LIN {X 0,Y 297.878,Z 251.743,A -85,B 0,C 180,E1 -16462.256,E2 -16462.256} C_VEL
LIN {X 0,Y 297.967,Z 251.372,A -85,B 0,C 180,E1 -16463.229,E2 -16463.229} C_VEL
LIN {X 0,Y 298.216,Z 251.337,A -85,B 0,C 180,E1 -16465.947,E2 -16465.947} C_VEL
LIN {X 0,Y 298.812,Z 251.261,A -85,B 0,C 180,E1 -16468.654,E2 -16468.654} C_VEL
LIN {X 0,Y 298.912,Z 251.253,A -85,B 0,C 180,E1 -16471.349,E2 -16471.349} C_VEL
LIN {X 0,Y 298.784,Z 251.266,A -85,B 0,C 180,E1 -16476.756,E2 -16476.756} C_VEL
LIN {X 0,Y 298.668,Z 251.281,A -85,B 0,C 180,E1 -16479.482,E2 -16479.482} C_VEL
LIN {X 0,Y 298.542,Z 251.295,A -85,B 0,C 180,E1 -16483.617,E2 -16483.617} C_VEL
LIN {X 0,Y 298.538,Z 251.296,A -85,B 0,C 180,E1 -16486.411,E2 -16486.411} C_VEL
LIN {X 0,Y 298.531,Z 251.297,A -85,B 0,C 180,E1 -16489.673,E2 -16489.673} C_VEL
LIN {X 0,Y 298.449,Z 251.307,A -85,B 0,C 180,E1 -16493.6,E2 -16493.6} C_VEL
LIN {X 0,Y 298.482,Z 251.306,A -85,B 0,C 180,E1 -16496.577,E2 -16496.577} C_VEL
LIN {X 0,Y 298.412,Z 251.312,A -85,B 0,C 180,E1 -16499.643,E2 -16499.643} C_VEL
LIN {X 0,Y 298.387,Z 251.319,A -85,B 0,C 180,E1 -16502.803,E2 -16502.803} C_VEL
LIN {X 0,Y 298.459,Z 251.309,A -85,B 0,C 180,E1 -16506.815,E2 -16506.815} C_VEL
LIN {X 0,Y 298.446,Z 251.307,A -85,B 0,C 180,E1 -16511.253,E2 -16511.253} C_VEL
LIN {X 0,Y 298.412,Z 251.311,A -85,B 0,C 180,E1 -16515.05,E2 -16515.05} C_VEL
LIN {X 0,Y 298.417,Z 251.313,A -85,B 0,C 180,E1 -16518.747,E2 -16518.747} C_VEL
LIN {X 0,Y 298.444,Z 251.309,A -85,B 0,C 180,E1 -16522.25,E2 -16522.25} C_VEL
LIN {X 0,Y 298.406,Z 251.307,A -85,B 0,C 180,E1 -16525.584,E2 -16525.584} C_VEL
LIN {X 0,Y 298.391,Z 251.314,A -85,B 0,C 180,E1 -16528.794,E2 -16528.794} C_VEL
LIN {X 0,Y 298.459,Z 251.307,A -85,B 0,C 180,E1 -16531.907,E2 -16531.907} C_VEL
LIN {X 0,Y 298.486,Z 251.301,A -85,B 0,C 180,E1 -16534.927,E2 -16534.927} C_VEL
LIN {X 0,Y 298.452,Z 251.301,A -85,B 0,C 180,E1 -16539.318,E2 -16539.318} C_VEL
LIN {X 0,Y 298.541,Z 251.297,A -85,B 0,C 180,E1 -16542.182,E2 -16542.182} C_VEL
LIN {X 0,Y 298.597,Z 251.287,A -85,B 0,C 180,E1 -16544.997,E2 -16544.997} C_VEL
LIN {X 0,Y 298.597,Z 251.287,A -85,B 0,C 180,E1 -16549.149,E2 -16549.149} C_VEL
LIN {X 0,Y 298.723,Z 251.274,A -85,B 0,C 180,E1 -16551.887,E2 -16551.887} C_VEL
LIN {X 0,Y 298.777,Z 251.262,A -85,B 0,C 180,E1 -16553.205,E2 -16553.205} C_VEL
LIN {X 0,Y 298.199,Z 251.337,A -85,B 0,C 180,E1 -16554.33,E2 -16554.33} C_VEL
LIN {X 0,Y 295.397,Z 251.687,A -85,B 0,C 180,E1 -16556.162,E2 -16556.162} C_VEL
LIN {X 0,Y 292.986,Z 251.988,A -85,B 0,C 180,E1 -16557.65,E2 -16557.65} C_VEL
LIN {X 0,Y 291.971,Z 252.112,A -85,B 0,C 180,E1 -16558.802,E2 -16558.802} C_VEL
LIN {X 0,Y 291.901,Z 252.12,A -85,B 0,C 180,E1 -16559.192,E2 -16559.192} C_VEL
LIN {X 0,Y 291.792,Z 252.135,A -85,B 0,C 180,E1 -16562.763,E2 -16562.763} C_VEL
LIN {X 0,Y 291.715,Z 252.142,A -85,B 0,C 180,E1 -16566.921,E2 -16566.921} C_VEL
LIN {X 0,Y 291.577,Z 252.165,A -85,B 0,C 180,E1 -16569.716,E2 -16569.716} C_VEL
LIN {X 0,Y 291.531,Z 252.17,A -85,B 0,C 180,E1 -16573.952,E2 -16573.952} C_VEL
LIN {X 0,Y 291.497,Z 252.172,A -85,B 0,C 180,E1 -16576.819,E2 -16576.819} C_VEL
LIN {X 0,Y 291.461,Z 252.177,A -85,B 0,C 180,E1 -16579.876,E2 -16579.876} C_VEL
LIN {X 0,Y 291.409,Z 252.183,A -85,B 0,C 180,E1 -16584.206,E2 -16584.206} C_VEL
LIN {X 0,Y 291.429,Z 252.183,A -85,B 0,C 180,E1 -16587.273,E2 -16587.273} C_VEL
LIN {X 0,Y 291.345,Z 252.191,A -85,B 0,C 180,E1 -16590.438,E2 -16590.438} C_VEL
LIN {X 0,Y 291.355,Z 252.191,A -85,B 0,C 180,E1 -16593.699,E2 -16593.699} C_VEL
LIN {X 0,Y 291.383,Z 252.19,A -85,B 0,C 180,E1 -16597.253,E2 -16597.253} C_VEL
LIN {X 0,Y 291.358,Z 252.193,A -85,B 0,C 180,E1 -16600.64,E2 -16600.64} C_VEL
LIN {X 0,Y 291.407,Z 252.343,A -85,B 0,C 180,E1 -16601.98,E2 -16601.98} C_VEL
LIN {X 0,Y 292.29,Z 257.456,A -85,B 0,C 180,E1 -16606.167,E2 -16606.167} C_VEL
LIN {X 0,Y 293.236,Z 262.543,A -85,B 0,C 180,E1 -16610.083,E2 -16610.083} C_VEL
LIN {X 0,Y 293.719,Z 266.92,A -85,B 0,C 180,E1 -16613.258,E2 -16613.258} C_VEL
LIN {X 0,Y 293.218,Z 270.535,A -85,B 0,C 180,E1 -16615.717,E2 -16615.717} C_VEL
LIN {X 0,Y 292.053,Z 277.114,A -85,B 0,C 180,E1 -16620.035,E2 -16620.035} C_VEL
LIN {X 0,Y 291.177,Z 283.685,A -85,B 0,C 180,E1 -16624.248,E2 -16624.248} C_VEL
LIN {X 0,Y 290.805,Z 286.658,A -85,B 0,C 180,E1 -16626.123,E2 -16626.123} C_VEL
LIN {X 0,Y 293.175,Z 300.593,A -85,B 0,C 180,E1 -16626.941,E2 -16626.941} C_VEL
LIN {X 0,Y 294.855,Z 313.515,A -85,B 0,C 180,E1 -16627.954,E2 -16627.954} C_VEL
LIN {X 0,Y 295.966,Z 325.481,A -85,B 0,C 180,E1 -16629.132,E2 -16629.132} C_VEL
LIN {X 0,Y 296.311,Z 334.899,A -85,B 0,C 180,E1 -16630.244,E2 -16630.244} C_VEL
LIN {X 0,Y 294.73,Z 346.056,A -85,B 0,C 180,E1 -16631.76,E2 -16631.76} C_VEL
LIN {X 0,Y 293.359,Z 355.626,A -85,B 0,C 180,E1 -16633.396,E2 -16633.396} C_VEL
LIN {X 0,Y 292.309,Z 363.424,A -85,B 0,C 180,E1 -16635.02,E2 -16635.02} C_VEL
LIN {X 0,Y 291.179,Z 371.571,A -85,B 0,C 180,E1 -16637.098,E2 -16637.098} C_VEL
LIN {X 0,Y 290.406,Z 377.096,A -85,B 0,C 180,E1 -16638.835,E2 -16638.835} C_VEL
LIN {X 0,Y 289.909,Z 382.504,A -85,B 0,C 180,E1 -16640.933,E2 -16640.933} C_VEL
LIN {X 0,Y 289.662,Z 386.705,A -85,B 0,C 180,E1 -16643.031,E2 -16643.031} C_VEL
LIN {X 0,Y 289.565,Z 388.913,A -85,B 0,C 180,E1 -16644.427,E2 -16644.427} C_VEL
LIN {X 0,Y 289.594,Z 390.629,A -85,B 0,C 180,E1 -16645.823,E2 -16645.823} C_VEL
LIN {X 0,Y 289.587,Z 391.918,A -85,B 0,C 180,E1 -16647.216,E2 -16647.216} C_VEL
LIN {X 0,Y 289.641,Z 392.803,A -85,B 0,C 180,E1 -16648.608,E2 -16648.608} C_VEL
LIN {X 0,Y 289.722,Z 393.271,A -85,B 0,C 180,E1 -16649.999,E2 -16649.999} C_VEL
LIN {X 0,Y 289.603,Z 393.288,A -85,B 0,C 180,E1 -16651.389,E2 -16651.389} C_VEL
LIN {X 0,Y 289.559,Z 392.914,A -85,B 0,C 180,E1 -16652.781,E2 -16652.781} C_VEL
LIN {X 0,Y 289.534,Z 392.146,A -85,B 0,C 180,E1 -16654.175,E2 -16654.175} C_VEL
LIN {X 0,Y 289.522,Z 390.972,A -85,B 0,C 180,E1 -16655.571,E2 -16655.571} C_VEL
LIN {X 0,Y 289.707,Z 388.403,A -85,B 0,C 180,E1 -16657.666,E2 -16657.666} C_VEL
LIN {X 0,Y 290.078,Z 384.831,A -85,B 0,C 180,E1 -16659.763,E2 -16659.763} C_VEL
LIN {X 0,Y 290.74,Z 380.19,A -85,B 0,C 180,E1 -16661.855,E2 -16661.855} C_VEL
LIN {X 0,Y 292.151,Z 373.245,A -85,B 0,C 180,E1 -16664.273,E2 -16664.273} C_VEL
LIN {X 0,Y 293.628,Z 365.768,A -85,B 0,C 180,E1 -16666.333,E2 -16666.333} C_VEL
LIN {X 0,Y 295.354,Z 356.558,A -85,B 0,C 180,E1 -16668.377,E2 -16668.377} C_VEL
LIN {X 0,Y 297.474,Z 346.002,A -85,B 0,C 180,E1 -16670.212,E2 -16670.212} C_VEL
LIN {X 0,Y 299.119,Z 336.644,A -85,B 0,C 180,E1 -16671.537,E2 -16671.537} C_VEL
LIN {X 0,Y 299.097,Z 325.654,A -85,B 0,C 180,E1 -16672.954,E2 -16672.954} C_VEL
LIN {X 0,Y 298.03,Z 313.134,A -85,B 0,C 180,E1 -16674.348,E2 -16674.348} C_VEL
LIN {X 0,Y 295.882,Z 300.736,A -85,B 0,C 180,E1 -16675.557,E2 -16675.557} C_VEL
LIN {X 0,Y 292.49,Z 287.558,A -85,B 0,C 180,E1 -16676.695,E2 -16676.695} C_VEL
LIN {X 0,Y 291.601,Z 284.162,A -85,B 0,C 180,E1 -16676.947,E2 -16676.947} C_VEL
LIN {X 0,Y 292.841,Z 276.861,A -85,B 0,C 180,E1 -16681.868,E2 -16681.868} C_VEL
LIN {X 0,Y 293.931,Z 271.595,A -85,B 0,C 180,E1 -16685.612,E2 -16685.612} C_VEL
LIN {X 0,Y 294.175,Z 270.188,A -85,B 0,C 180,E1 -16686.672,E2 -16686.672} C_VEL
LIN {X 0,Y 294.068,Z 267.992,A -85,B 0,C 180,E1 -16688.415,E2 -16688.415} C_VEL
LIN {X 0,Y 293.408,Z 263.727,A -85,B 0,C 180,E1 -16692.118,E2 -16692.118} C_VEL
LIN {X 0,Y 292.651,Z 259.608,A -85,B 0,C 180,E1 -16696.089,E2 -16696.089} C_VEL
LIN {X 0,Y 291.977,Z 255.678,A -85,B 0,C 180,E1 -16700.374,E2 -16700.374} C_VEL
LIN {X 0,Y 291.629,Z 253.619,A -85,B 0,C 180,E1 -16702.95,E2 -16702.95} C_VEL
LIN {X 0,Y 291.369,Z 252.194,A -85,B 0,C 180,E1 -16705.092,E2 -16705.092} C_VEL
LIN {X 0,Y 291.371,Z 252.194,A -85,B 0,C 180,E1 -16707.949,E2 -16707.949} C_VEL
LIN {X 0,Y 291.38,Z 252.191,A -85,B 0,C 180,E1 -16711.156,E2 -16711.156} C_VEL
LIN {X 0,Y 291.414,Z 252.187,A -85,B 0,C 180,E1 -16714.27,E2 -16714.27} C_VEL
LIN {X 0,Y 291.379,Z 252.19,A -85,B 0,C 180,E1 -16717.297,E2 -16717.297} C_VEL
LIN {X 0,Y 291.455,Z 252.18,A -85,B 0,C 180,E1 -16720.268,E2 -16720.268} C_VEL
LIN {X 0,Y 291.551,Z 252.168,A -85,B 0,C 180,E1 -16724.621,E2 -16724.621} C_VEL
LIN {X 0,Y 291.534,Z 252.171,A -85,B 0,C 180,E1 -16728.878,E2 -16728.878} C_VEL
LIN {X 0,Y 291.704,Z 252.15,A -85,B 0,C 180,E1 -16731.686,E2 -16731.686} C_VEL
LIN {X 0,Y 291.627,Z 252.159,A -85,B 0,C 180,E1 -16734.466,E2 -16734.466} C_VEL
LIN {X 0,Y 291.884,Z 252.128,A -85,B 0,C 180,E1 -16738.618,E2 -16738.618} C_VEL
LIN {X 0,Y 291.885,Z 252.128,A -85,B 0,C 180,E1 -16741.378,E2 -16741.378} C_VEL
LIN {X 0,Y 291.739,Z 252.143,A -85,B 0,C 180,E1 -16746.916,E2 -16746.916} C_VEL
LIN {X 0,Y 291.621,Z 252.162,A -85,B 0,C 180,E1 -16749.71,E2 -16749.71} C_VEL
LIN {X 0,Y 291.504,Z 252.179,A -85,B 0,C 180,E1 -16753.949,E2 -16753.949} C_VEL
LIN {X 0,Y 291.548,Z 253.73,A -85,B 0,C 180,E1 -16756.812,E2 -16756.812} C_VEL
LIN {X 0,Y 291.501,Z 255.573,A -85,B 0,C 180,E1 -16759.906,E2 -16759.906} C_VEL
LIN {X 0,Y 291.255,Z 257.883,A -85,B 0,C 180,E1 -16763.521,E2 -16763.521} C_VEL
LIN {X 0,Y 291.048,Z 259.624,A -85,B 0,C 180,E1 -16766.095,E2 -16766.095} C_VEL
LIN {X 0,Y 292.201,Z 262.851,A -85,B 0,C 180,E1 -16766.414,E2 -16766.414} C_VEL
LIN {X 0,Y 296.691,Z 274.182,A -85,B 0,C 180,E1 -16767.651,E2 -16767.651} C_VEL
LIN {X 0,Y 299.912,Z 284.645,A -85,B 0,C 180,E1 -16768.88,E2 -16768.88} C_VEL
LIN {X 0,Y 302.255,Z 295.27,A -85,B 0,C 180,E1 -16770.242,E2 -16770.242} C_VEL
LIN {X 0,Y 302.598,Z 297.676,A -85,B 0,C 180,E1 -16770.569,E2 -16770.569} C_VEL
LIN {X 0,Y 300.991,Z 308.423,A -85,B 0,C 180,E1 -16771.863,E2 -16771.863} C_VEL
LIN {X 0,Y 299.09,Z 319.099,A -85,B 0,C 180,E1 -16773.472,E2 -16773.472} C_VEL
LIN {X 0,Y 297.172,Z 328.8,A -85,B 0,C 180,E1 -16775.325,E2 -16775.325} C_VEL
LIN {X 0,Y 295.453,Z 336.613,A -85,B 0,C 180,E1 -16777.17,E2 -16777.17} C_VEL
LIN {X 0,Y 293.915,Z 343.386,A -85,B 0,C 180,E1 -16779.153,E2 -16779.153} C_VEL
LIN {X 0,Y 292.712,Z 348.623,A -85,B 0,C 180,E1 -16781.07,E2 -16781.07} C_VEL
LIN {X 0,Y 291.737,Z 352.849,A -85,B 0,C 180,E1 -16783.018,E2 -16783.018} C_VEL
LIN {X 0,Y 290.734,Z 356.874,A -85,B 0,C 180,E1 -16785.493,E2 -16785.493} C_VEL
LIN {X 0,Y 290.171,Z 358.907,A -85,B 0,C 180,E1 -16787.302,E2 -16787.302} C_VEL
LIN {X 0,Y 289.823,Z 360.236,A -85,B 0,C 180,E1 -16789.103,E2 -16789.103} C_VEL
LIN {X 0,Y 289.581,Z 360.934,A -85,B 0,C 180,E1 -16790.948,E2 -16790.948} C_VEL
LIN {X 0,Y 289.434,Z 360.798,A -85,B 0,C 180,E1 -16793.25,E2 -16793.25} C_VEL
LIN {X 0,Y 289.574,Z 359.526,A -85,B 0,C 180,E1 -16795.602,E2 -16795.602} C_VEL
LIN {X 0,Y 289.895,Z 356.973,A -85,B 0,C 180,E1 -16798.045,E2 -16798.045} C_VEL
LIN {X 0,Y 290.474,Z 352.938,A -85,B 0,C 180,E1 -16800.571,E2 -16800.571} C_VEL
LIN {X 0,Y 291.068,Z 348.315,A -85,B 0,C 180,E1 -16802.694,E2 -16802.694} C_VEL
LIN {X 0,Y 291.918,Z 342.744,A -85,B 0,C 180,E1 -16804.703,E2 -16804.703} C_VEL
LIN {X 0,Y 292.962,Z 335.902,A -85,B 0,C 180,E1 -16806.684,E2 -16806.684} C_VEL
LIN {X 0,Y 294.217,Z 327.347,A -85,B 0,C 180,E1 -16808.677,E2 -16808.677} C_VEL
LIN {X 0,Y 295.76,Z 317.21,A -85,B 0,C 180,E1 -16810.57,E2 -16810.57} C_VEL
LIN {X 0,Y 297.122,Z 306.976,A -85,B 0,C 180,E1 -16812.093,E2 -16812.093} C_VEL
LIN {X 0,Y 298.379,Z 295.987,A -85,B 0,C 180,E1 -16813.407,E2 -16813.407} C_VEL
LIN {X 0,Y 298.756,Z 292.354,A -85,B 0,C 180,E1 -16813.78,E2 -16813.78} C_VEL
LIN {X 0,Y 296.429,Z 280.089,A -85,B 0,C 180,E1 -16815.065,E2 -16815.065} C_VEL
LIN {X 0,Y 293.36,Z 267.572,A -85,B 0,C 180,E1 -16816.14,E2 -16816.14} C_VEL
LIN {X 0,Y 290.474,Z 257.017,A -85,B 0,C 180,E1 -16816.891,E2 -16816.891} C_VEL
LIN {X 0,Y 290.734,Z 253.095,A -85,B 0,C 180,E1 -16821.662,E2 -16821.662} C_VEL
LIN {X 0,Y 290.89,Z 252.254,A -85,B 0,C 180,E1 -16823.063,E2 -16823.063} C_VEL
LIN {X 0,Y 291.164,Z 252.216,A -85,B 0,C 180,E1 -16825.849,E2 -16825.849} C_VEL
LIN {X 0,Y 291.768,Z 252.139,A -85,B 0,C 180,E1 -16828.621,E2 -16828.621} C_VEL
LIN {X 0,Y 291.878,Z 252.129,A -85,B 0,C 180,E1 -16831.381,E2 -16831.381} C_VEL
LIN {X 0,Y 291.733,Z 252.145,A -85,B 0,C 180,E1 -16836.92,E2 -16836.92} C_VEL
LIN {X 0,Y 291.617,Z 252.158,A -85,B 0,C 180,E1 -16839.714,E2 -16839.714} C_VEL
LIN {X 0,Y 291.511,Z 252.169,A -85,B 0,C 180,E1 -16843.952,E2 -16843.952} C_VEL
LIN {X 0,Y 291.477,Z 252.178,A -85,B 0,C 180,E1 -16846.82,E2 -16846.82} C_VEL
LIN {X 0,Y 291.473,Z 252.176,A -85,B 0,C 180,E1 -16849.895,E2 -16849.895} C_VEL
LIN {X 0,Y 291.392,Z 252.186,A -85,B 0,C 180,E1 -16854.207,E2 -16854.207} C_VEL
LIN {X 0,Y 291.416,Z 252.185,A -85,B 0,C 180,E1 -16857.274,E2 -16857.274} C_VEL
LIN {X 0,Y 291.329,Z 252.196,A -85,B 0,C 180,E1 -16860.439,E2 -16860.439} C_VEL
LIN {X 0,Y 291.337,Z 252.192,A -85,B 0,C 180,E1 -16863.701,E2 -16863.701} C_VEL
LIN {X 0,Y 291.392,Z 252.187,A -85,B 0,C 180,E1 -16867.263,E2 -16867.263} C_VEL
LIN {X 0,Y 291.395,Z 252.189,A -85,B 0,C 180,E1 -16870.634,E2 -16870.634} C_VEL
LIN {X 0,Y 291.348,Z 252.194,A -85,B 0,C 180,E1 -16874.393,E2 -16874.393} C_VEL
LIN {X 0,Y 291.354,Z 252.194,A -85,B 0,C 180,E1 -16878.4,E2 -16878.4} C_VEL
LIN {X 0,Y 291.378,Z 252.186,A -85,B 0,C 180,E1 -16881.166,E2 -16881.166} C_VEL
LIN {X 0,Y 291.384,Z 252.183,A -85,B 0,C 180,E1 -16884.633,E2 -16884.633} C_VEL
LIN {X 0,Y 291.369,Z 252.187,A -85,B 0,C 180,E1 -16887.953,E2 -16887.953} C_VEL
LIN {X 0,Y 291.377,Z 252.187,A -85,B 0,C 180,E1 -16891.161,E2 -16891.161} C_VEL
LIN {X 0,Y 291.416,Z 252.186,A -85,B 0,C 180,E1 -16894.275,E2 -16894.275} C_VEL
LIN {X 0,Y 291.383,Z 252.184,A -85,B 0,C 180,E1 -16897.302,E2 -16897.302} C_VEL
LIN {X 0,Y 291.461,Z 252.176,A -85,B 0,C 180,E1 -16900.273,E2 -16900.273} C_VEL
LIN {X 0,Y 291.559,Z 252.165,A -85,B 0,C 180,E1 -16904.626,E2 -16904.626} C_VEL
LIN {X 0,Y 291.541,Z 252.166,A -85,B 0,C 180,E1 -16908.883,E2 -16908.883} C_VEL
LIN {X 0,Y 291.673,Z 252.152,A -85,B 0,C 180,E1 -16911.69,E2 -16911.69} C_VEL
LIN {X 0,Y 291.629,Z 252.151,A -85,B 0,C 180,E1 -16914.471,E2 -16914.471} C_VEL
LIN {X 0,Y 291.895,Z 252.122,A -85,B 0,C 180,E1 -16918.623,E2 -16918.623} C_VEL
LIN {X 0,Y 291.901,Z 252.12,A -85,B 0,C 180,E1 -16919.192,E2 -16919.192} C_VEL
LIN {X 0,Y 291.59,Z 252.164,A -85,B 0,C 180,E1 -16919.962,E2 -16919.962} C_VEL
LIN {X 0,Y 290.177,Z 252.339,A -85,B 0,C 180,E1 -16921.096,E2 -16921.096} C_VEL
LIN {X 0,Y 285.646,Z 252.904,A -85,B 0,C 180,E1 -16923.731,E2 -16923.731} C_VEL
LIN {X 0,Y 284.607,Z 253.029,A -85,B 0,C 180,E1 -16924.912,E2 -16924.912} C_VEL
LIN {X 0,Y 284.553,Z 253.035,A -85,B 0,C 180,E1 -16925.312,E2 -16925.312} C_VEL
LIN {X 0,Y 284.63,Z 253.024,A -85,B 0,C 180,E1 -16928.522,E2 -16928.522} C_VEL
LIN {X 0,Y 284.484,Z 253.046,A -85,B 0,C 180,E1 -16932.849,E2 -16932.849} C_VEL
LIN {X 0,Y 284.497,Z 253.046,A -85,B 0,C 180,E1 -16935.77,E2 -16935.77} C_VEL
LIN {X 0,Y 284.389,Z 253.056,A -85,B 0,C 180,E1 -16940.244,E2 -16940.244} C_VEL
LIN {X 0,Y 284.379,Z 253.06,A -85,B 0,C 180,E1 -16943.876,E2 -16943.876} C_VEL
LIN {X 0,Y 284.405,Z 253.058,A -85,B 0,C 180,E1 -16947.173,E2 -16947.173} C_VEL
LIN {X 0,Y 284.304,Z 253.073,A -85,B 0,C 180,E1 -16951.275,E2 -16951.275} C_VEL
LIN {X 0,Y 284.351,Z 253.065,A -85,B 0,C 180,E1 -16955.349,E2 -16955.349} C_VEL
LIN {X 0,Y 284.319,Z 253.066,A -85,B 0,C 180,E1 -16958.17,E2 -16958.17} C_VEL
LIN {X 0,Y 284.37,Z 253.201,A -85,B 0,C 180,E1 -16961.623,E2 -16961.623} C_VEL
LIN {X 0,Y 285.156,Z 257.944,A -85,B 0,C 180,E1 -16965.624,E2 -16965.624} C_VEL
LIN {X 0,Y 286.115,Z 262.952,A -85,B 0,C 180,E1 -16969.596,E2 -16969.596} C_VEL
LIN {X 0,Y 286.675,Z 267.618,A -85,B 0,C 180,E1 -16973.083,E2 -16973.083} C_VEL
LIN {X 0,Y 286.2,Z 271.238,A -85,B 0,C 180,E1 -16975.61,E2 -16975.61} C_VEL
LIN {X 0,Y 284.88,Z 278.396,A -85,B 0,C 180,E1 -16980.434,E2 -16980.434} C_VEL
LIN {X 0,Y 284.065,Z 284.332,A -85,B 0,C 180,E1 -16984.343,E2 -16984.343} C_VEL
LIN {X 0,Y 283.82,Z 286.254,A -85,B 0,C 180,E1 -16985.591,E2 -16985.591} C_VEL
LIN {X 0,Y 286.285,Z 300.737,A -85,B 0,C 180,E1 -16986.494,E2 -16986.494} C_VEL
LIN {X 0,Y 288.003,Z 314.305,A -85,B 0,C 180,E1 -16987.606,E2 -16987.606} C_VEL
LIN {X 0,Y 289.03,Z 325.864,A -85,B 0,C 180,E1 -16988.794,E2 -16988.794} C_VEL
LIN {X 0,Y 289.403,Z 335.147,A -85,B 0,C 180,E1 -16989.938,E2 -16989.938} C_VEL
LIN {X 0,Y 287.773,Z 346.146,A -85,B 0,C 180,E1 -16991.488,E2 -16991.488} C_VEL
LIN {X 0,Y 286.353,Z 355.715,A -85,B 0,C 180,E1 -16993.178,E2 -16993.178} C_VEL
LIN {X 0,Y 285.156,Z 364.113,A -85,B 0,C 180,E1 -16995.001,E2 -16995.001} C_VEL
LIN {X 0,Y 284.036,Z 372.066,A -85,B 0,C 180,E1 -16997.131,E2 -16997.131} C_VEL
LIN {X 0,Y 283.186,Z 378.4,A -85,B 0,C 180,E1 -16999.271,E2 -16999.271} C_VEL
LIN {X 0,Y 282.756,Z 383.437,A -85,B 0,C 180,E1 -17001.422,E2 -17001.422} C_VEL
LIN {X 0,Y 282.538,Z 387.312,A -85,B 0,C 180,E1 -17003.572,E2 -17003.572} C_VEL
LIN {X 0,Y 282.508,Z 390.131,A -85,B 0,C 180,E1 -17005.719,E2 -17005.719} C_VEL
LIN {X 0,Y 282.512,Z 391.443,A -85,B 0,C 180,E1 -17007.147,E2 -17007.147} C_VEL
LIN {X 0,Y 282.552,Z 392.348,A -85,B 0,C 180,E1 -17008.573,E2 -17008.573} C_VEL
LIN {X 0,Y 282.632,Z 392.851,A -85,B 0,C 180,E1 -17009.999,E2 -17009.999} C_VEL
LIN {X 0,Y 282.516,Z 392.895,A -85,B 0,C 180,E1 -17011.424,E2 -17011.424} C_VEL
LIN {X 0,Y 282.483,Z 392.541,A -85,B 0,C 180,E1 -17012.851,E2 -17012.851} C_VEL
LIN {X 0,Y 282.428,Z 390.827,A -85,B 0,C 180,E1 -17015.502,E2 -17015.502} C_VEL
LIN {X 0,Y 282.638,Z 388.111,A -85,B 0,C 180,E1 -17017.859,E2 -17017.859} C_VEL
LIN {X 0,Y 283.061,Z 384.593,A -85,B 0,C 180,E1 -17020.007,E2 -17020.007} C_VEL
LIN {X 0,Y 283.762,Z 380.014,A -85,B 0,C 180,E1 -17022.151,E2 -17022.151} C_VEL
LIN {X 0,Y 285.265,Z 373.162,A -85,B 0,C 180,E1 -17024.626,E2 -17024.626} C_VEL
LIN {X 0,Y 286.813,Z 365.752,A -85,B 0,C 180,E1 -17026.732,E2 -17026.732} C_VEL
LIN {X 0,Y 288.603,Z 356.636,A -85,B 0,C 180,E1 -17028.822,E2 -17028.822} C_VEL
LIN {X 0,Y 290.821,Z 346.209,A -85,B 0,C 180,E1 -17030.696,E2 -17030.696} C_VEL
LIN {X 0,Y 292.377,Z 338.261,A -85,B 0,C 180,E1 -17031.873,E2 -17031.873} C_VEL
LIN {X 0,Y 292.578,Z 328.257,A -85,B 0,C 180,E1 -17033.249,E2 -17033.249} C_VEL
LIN {X 0,Y 291.762,Z 315.977,A -85,B 0,C 180,E1 -17034.721,E2 -17034.721} C_VEL
LIN {X 0,Y 289.917,Z 304.046,A -85,B 0,C 180,E1 -17035.982,E2 -17035.982} C_VEL
LIN {X 0,Y 286.778,Z 290.743,A -85,B 0,C 180,E1 -17037.233,E2 -17037.233} C_VEL
LIN {X 0,Y 284.767,Z 284.329,A -85,B 0,C 180,E1 -17037.8,E2 -17037.8} C_VEL
LIN {X 0,Y 284.701,Z 283.664,A -85,B 0,C 180,E1 -17037.859,E2 -17037.859} C_VEL
LIN {X 0,Y 286.016,Z 276.704,A -85,B 0,C 180,E1 -17042.722,E2 -17042.722} C_VEL
LIN {X 0,Y 287.007,Z 272.147,A -85,B 0,C 180,E1 -17046.089,E2 -17046.089} C_VEL
LIN {X 0,Y 287.143,Z 270.064,A -85,B 0,C 180,E1 -17047.724,E2 -17047.724} C_VEL
LIN {X 0,Y 286.555,Z 265.789,A -85,B 0,C 180,E1 -17051.466,E2 -17051.466} C_VEL
LIN {X 0,Y 285.782,Z 261.651,A -85,B 0,C 180,E1 -17055.491,E2 -17055.491} C_VEL
LIN {X 0,Y 285.334,Z 259.033,A -85,B 0,C 180,E1 -17058.313,E2 -17058.313} C_VEL
LIN {X 0,Y 284.836,Z 255.837,A -85,B 0,C 180,E1 -17062.142,E2 -17062.142} C_VEL
LIN {X 0,Y 284.39,Z 253.529,A -85,B 0,C 180,E1 -17065.36,E2 -17065.36} C_VEL
LIN {X 0,Y 284.307,Z 253.073,A -85,B 0,C 180,E1 -17067.187,E2 -17067.187} C_VEL
LIN {X 0,Y 284.357,Z 253.067,A -85,B 0,C 180,E1 -17070.374,E2 -17070.374} C_VEL
LIN {X 0,Y 284.376,Z 253.063,A -85,B 0,C 180,E1 -17073.584,E2 -17073.584} C_VEL
LIN {X 0,Y 284.364,Z 253.066,A -85,B 0,C 180,E1 -17076.705,E2 -17076.705} C_VEL
LIN {X 0,Y 284.4,Z 253.059,A -85,B 0,C 180,E1 -17081.259,E2 -17081.259} C_VEL
LIN {X 0,Y 284.488,Z 253.047,A -85,B 0,C 180,E1 -17084.457,E2 -17084.457} C_VEL
LIN {X 0,Y 284.486,Z 253.048,A -85,B 0,C 180,E1 -17088.599,E2 -17088.599} C_VEL
LIN {X 0,Y 284.654,Z 253.028,A -85,B 0,C 180,E1 -17091.479,E2 -17091.479} C_VEL
LIN {X 0,Y 284.597,Z 253.035,A -85,B 0,C 180,E1 -17094.329,E2 -17094.329} C_VEL
LIN {X 0,Y 284.85,Z 253.004,A -85,B 0,C 180,E1 -17098.584,E2 -17098.584} C_VEL
LIN {X 0,Y 284.851,Z 253.004,A -85,B 0,C 180,E1 -17101.412,E2 -17101.412} C_VEL
LIN {X 0,Y 284.691,Z 253.021,A -85,B 0,C 180,E1 -17107.088,E2 -17107.088} C_VEL
LIN {X 0,Y 284.559,Z 253.04,A -85,B 0,C 180,E1 -17109.953,E2 -17109.953} C_VEL
LIN {X 0,Y 284.465,Z 253.053,A -85,B 0,C 180,E1 -17112.845,E2 -17112.845} C_VEL
LIN {X 0,Y 284.56,Z 254.408,A -85,B 0,C 180,E1 -17115.761,E2 -17115.761} C_VEL
LIN {X 0,Y 284.554,Z 256.055,A -85,B 0,C 180,E1 -17118.726,E2 -17118.726} C_VEL
LIN {X 0,Y 284.335,Z 257.92,A -85,B 0,C 180,E1 -17121.76,E2 -17121.76} C_VEL
LIN {X 0,Y 284.082,Z 260.226,A -85,B 0,C 180,E1 -17125.21,E2 -17125.21} C_VEL
LIN {X 0,Y 285.279,Z 263.405,A -85,B 0,C 180,E1 -17125.536,E2 -17125.536} C_VEL
LIN {X 0,Y 289.603,Z 273.829,A -85,B 0,C 180,E1 -17126.761,E2 -17126.761} C_VEL
LIN {X 0,Y 293.122,Z 284.677,A -85,B 0,C 180,E1 -17128.103,E2 -17128.103} C_VEL
LIN {X 0,Y 295.569,Z 295.709,A -85,B 0,C 180,E1 -17129.561,E2 -17129.561} C_VEL
LIN {X 0,Y 296.129,Z 299.137,A -85,B 0,C 180,E1 -17130.053,E2 -17130.053} C_VEL
LIN {X 0,Y 294.431,Z 309.949,A -85,B 0,C 180,E1 -17131.414,E2 -17131.414} C_VEL
LIN {X 0,Y 292.43,Z 320.362,A -85,B 0,C 180,E1 -17133.06,E2 -17133.06} C_VEL
LIN {X 0,Y 290.435,Z 329.954,A -85,B 0,C 180,E1 -17134.964,E2 -17134.964} C_VEL
LIN {X 0,Y 288.613,Z 337.763,A -85,B 0,C 180,E1 -17136.88,E2 -17136.88} C_VEL
LIN {X 0,Y 286.847,Z 344.951,A -85,B 0,C 180,E1 -17139.111,E2 -17139.111} C_VEL
LIN {X 0,Y 285.284,Z 351.331,A -85,B 0,C 180,E1 -17141.69,E2 -17141.69} C_VEL
LIN {X 0,Y 284.116,Z 355.828,A -85,B 0,C 180,E1 -17144.166,E2 -17144.166} C_VEL
LIN {X 0,Y 283.477,Z 358.296,A -85,B 0,C 180,E1 -17146.04,E2 -17146.04} C_VEL
LIN {X 0,Y 282.904,Z 360.21,A -85,B 0,C 180,E1 -17148.178,E2 -17148.178} C_VEL
LIN {X 0,Y 282.535,Z 361.253,A -85,B 0,C 180,E1 -17150.45,E2 -17150.45} C_VEL
LIN {X 0,Y 282.368,Z 361.142,A -85,B 0,C 180,E1 -17153.322,E2 -17153.322} C_VEL
LIN {X 0,Y 282.442,Z 360.211,A -85,B 0,C 180,E1 -17155.194,E2 -17155.194} C_VEL
LIN {X 0,Y 282.74,Z 357.885,A -85,B 0,C 180,E1 -17157.68,E2 -17157.68} C_VEL
LIN {X 0,Y 283.309,Z 354.064,A -85,B 0,C 180,E1 -17160.257,E2 -17160.257} C_VEL
LIN {X 0,Y 283.908,Z 349.509,A -85,B 0,C 180,E1 -17162.495,E2 -17162.495} C_VEL
LIN {X 0,Y 284.867,Z 343.382,A -85,B 0,C 180,E1 -17164.814,E2 -17164.814} C_VEL
LIN {X 0,Y 285.933,Z 336.614,A -85,B 0,C 180,E1 -17166.844,E2 -17166.844} C_VEL
LIN {X 0,Y 287.24,Z 328.14,A -85,B 0,C 180,E1 -17168.88,E2 -17168.88} C_VEL
LIN {X 0,Y 288.792,Z 318.404,A -85,B 0,C 180,E1 -17170.76,E2 -17170.76} C_VEL
LIN {X 0,Y 290.241,Z 307.938,A -85,B 0,C 180,E1 -17172.383,E2 -17172.383} C_VEL
LIN {X 0,Y 291.546,Z 297.063,A -85,B 0,C 180,E1 -17173.727,E2 -17173.727} C_VEL
LIN {X 0,Y 291.925,Z 293.518,A -85,B 0,C 180,E1 -17174.108,E2 -17174.108} C_VEL
LIN {X 0,Y 289.666,Z 281.484,A -85,B 0,C 180,E1 -17175.422,E2 -17175.422} C_VEL
LIN {X 0,Y 286.527,Z 268.683,A -85,B 0,C 180,E1 -17176.572,E2 -17176.572} C_VEL
LIN {X 0,Y 283.415,Z 257.418,A -85,B 0,C 180,E1 -17177.379,E2 -17177.379} C_VEL
LIN {X 0,Y 283.751,Z 253.539,A -85,B 0,C 180,E1 -17182.17,E2 -17182.17} C_VEL
LIN {X 0,Y 283.815,Z 253.136,A -85,B 0,C 180,E1 -17182.889,E2 -17182.889} C_VEL
LIN {X 0,Y 284.112,Z 253.095,A -85,B 0,C 180,E1 -17185.746,E2 -17185.746} C_VEL
LIN {X 0,Y 284.723,Z 253.016,A -85,B 0,C 180,E1 -17188.587,E2 -17188.587} C_VEL
LIN {X 0,Y 284.844,Z 253.005,A -85,B 0,C 180,E1 -17191.415,E2 -17191.415} C_VEL
LIN {X 0,Y 284.685,Z 253.025,A -85,B 0,C 180,E1 -17197.092,E2 -17197.092} C_VEL
LIN {X 0,Y 284.555,Z 253.037,A -85,B 0,C 180,E1 -17199.957,E2 -17199.957} C_VEL
LIN {X 0,Y 284.471,Z 253.046,A -85,B 0,C 180,E1 -17204.305,E2 -17204.305} C_VEL
LIN {X 0,Y 284.418,Z 253.059,A -85,B 0,C 180,E1 -17207.25,E2 -17207.25} C_VEL
LIN {X 0,Y 284.409,Z 253.056,A -85,B 0,C 180,E1 -17210.241,E2 -17210.241} C_VEL
LIN {X 0,Y 284.361,Z 253.062,A -85,B 0,C 180,E1 -17213.878,E2 -17213.878} C_VEL
LIN {X 0,Y 284.39,Z 253.061,A -85,B 0,C 180,E1 -17217.177,E2 -17217.177} C_VEL
LIN {X 0,Y 284.287,Z 253.073,A -85,B 0,C 180,E1 -17221.277,E2 -17221.277} C_VEL
LIN {X 0,Y 284.354,Z 253.063,A -85,B 0,C 180,E1 -17225.357,E2 -17225.357} C_VEL
LIN {X 0,Y 284.325,Z 253.067,A -85,B 0,C 180,E1 -17228.169,E2 -17228.169} C_VEL
LIN {X 0,Y 284.335,Z 253.066,A -85,B 0,C 180,E1 -17232.143,E2 -17232.143} C_VEL
LIN {X 0,Y 284.314,Z 253.068,A -85,B 0,C 180,E1 -17236.204,E2 -17236.204} C_VEL
LIN {X 0,Y 284.348,Z 253.064,A -85,B 0,C 180,E1 -17240.016,E2 -17240.016} C_VEL
LIN {X 0,Y 284.353,Z 253.059,A -85,B 0,C 180,E1 -17243.62,E2 -17243.62} C_VEL
LIN {X 0,Y 284.306,Z 253.064,A -85,B 0,C 180,E1 -17247.193,E2 -17247.193} C_VEL
LIN {X 0,Y 284.355,Z 253.066,A -85,B 0,C 180,E1 -17250.379,E2 -17250.379} C_VEL
LIN {X 0,Y 284.377,Z 253.06,A -85,B 0,C 180,E1 -17253.589,E2 -17253.589} C_VEL
LIN {X 0,Y 284.368,Z 253.058,A -85,B 0,C 180,E1 -17256.71,E2 -17256.71} C_VEL
LIN {X 0,Y 284.406,Z 253.05,A -85,B 0,C 180,E1 -17261.264,E2 -17261.264} C_VEL
LIN {X 0,Y 284.496,Z 253.045,A -85,B 0,C 180,E1 -17264.462,E2 -17264.462} C_VEL
LIN {X 0,Y 284.493,Z 253.045,A -85,B 0,C 180,E1 -17268.604,E2 -17268.604} C_VEL
LIN {X 0,Y 284.627,Z 253.027,A -85,B 0,C 180,E1 -17271.483,E2 -17271.483} C_VEL
LIN {X 0,Y 284.598,Z 253.027,A -85,B 0,C 180,E1 -17274.333,E2 -17274.333} C_VEL
LIN {X 0,Y 284.861,Z 252.998,A -85,B 0,C 180,E1 -17278.588,E2 -17278.588} C_VEL
LIN {X 0,Y 284.861,Z 253.001,A -85,B 0,C 180,E1 -17281.416,E2 -17281.416} C_VEL
LIN {X 0,Y 284.553,Z 253.035,A -85,B 0,C 180,E1 -17285.312,E2 -17285.312} C_VEL
LIN {X 0,Y 284.29,Z 253.071,A -85,B 0,C 180,E1 -17286.103,E2 -17286.103} C_VEL
LIN {X 0,Y 282.958,Z 253.236,A -85,B 0,C 180,E1 -17287.269,E2 -17287.269} C_VEL
LIN {X 0,Y 278.556,Z 253.785,A -85,B 0,C 180,E1 -17289.981,E2 -17289.981} C_VEL
LIN {X 0,Y 277.507,Z 253.915,A -85,B 0,C 180,E1 -17291.194,E2 -17291.194} C_VEL
LIN {X 0,Y 277.436,Z 253.927,A -85,B 0,C 180,E1 -17291.606,E2 -17291.606} C_VEL
LIN {X 0,Y 277.453,Z 253.923,A -85,B 0,C 180,E1 -17295.724,E2 -17295.724} C_VEL
LIN {X 0,Y 277.355,Z 253.932,A -85,B 0,C 180,E1 -17300.351,E2 -17300.351} C_VEL
LIN {X 0,Y 277.329,Z 253.938,A -85,B 0,C 180,E1 -17304.171,E2 -17304.171} C_VEL
LIN {X 0,Y 277.333,Z 253.937,A -85,B 0,C 180,E1 -17307.505,E2 -17307.505} C_VEL
LIN {X 0,Y 277.283,Z 253.943,A -85,B 0,C 180,E1 -17310.482,E2 -17310.482} C_VEL
LIN {X 0,Y 277.257,Z 253.946,A -85,B 0,C 180,E1 -17313.896,E2 -17313.896} C_VEL
LIN {X 0,Y 277.275,Z 253.946,A -85,B 0,C 180,E1 -17317.47,E2 -17317.47} C_VEL
LIN {X 0,Y 277.301,Z 254.025,A -85,B 0,C 180,E1 -17321.222,E2 -17321.222} C_VEL
LIN {X 0,Y 278.038,Z 258.43,A -85,B 0,C 180,E1 -17325.055,E2 -17325.055} C_VEL
LIN {X 0,Y 278.965,Z 263.364,A -85,B 0,C 180,E1 -17329.097,E2 -17329.097} C_VEL
LIN {X 0,Y 279.549,Z 267.195,A -85,B 0,C 180,E1 -17332.084,E2 -17332.084} C_VEL
LIN {X 0,Y 279.366,Z 270.698,A -85,B 0,C 180,E1 -17334.646,E2 -17334.646} C_VEL
LIN {X 0,Y 278.424,Z 275.472,A -85,B 0,C 180,E1 -17337.987,E2 -17337.987} C_VEL
LIN {X 0,Y 277.343,Z 282.061,A -85,B 0,C 180,E1 -17342.491,E2 -17342.491} C_VEL
LIN {X 0,Y 276.842,Z 285.927,A -85,B 0,C 180,E1 -17345.086,E2 -17345.086} C_VEL
LIN {X 0,Y 279.238,Z 299.838,A -85,B 0,C 180,E1 -17345.958,E2 -17345.958} C_VEL
LIN {X 0,Y 280.974,Z 312.957,A -85,B 0,C 180,E1 -17347.05,E2 -17347.05} C_VEL
LIN {X 0,Y 281.971,Z 324.437,A -85,B 0,C 180,E1 -17348.237,E2 -17348.237} C_VEL
LIN {X 0,Y 282.474,Z 335.386,A -85,B 0,C 180,E1 -17349.614,E2 -17349.614} C_VEL
LIN {X 0,Y 280.817,Z 346.234,A -85,B 0,C 180,E1 -17351.201,E2 -17351.201} C_VEL
LIN {X 0,Y 279.374,Z 355.725,A -85,B 0,C 180,E1 -17352.933,E2 -17352.933} C_VEL
LIN {X 0,Y 278.005,Z 364.797,A -85,B 0,C 180,E1 -17354.981,E2 -17354.981} C_VEL
LIN {X 0,Y 276.871,Z 372.491,A -85,B 0,C 180,E1 -17357.166,E2 -17357.166} C_VEL
LIN {X 0,Y 275.98,Z 379.582,A -85,B 0,C 180,E1 -17359.73,E2 -17359.73} C_VEL
LIN {X 0,Y 275.59,Z 384.28,A -85,B 0,C 180,E1 -17361.936,E2 -17361.936} C_VEL
LIN {X 0,Y 275.451,Z 388.095,A -85,B 0,C 180,E1 -17364.321,E2 -17364.321} C_VEL
LIN {X 0,Y 275.429,Z 389.635,A -85,B 0,C 180,E1 -17365.608,E2 -17365.608} C_VEL
LIN {X 0,Y 275.438,Z 390.968,A -85,B 0,C 180,E1 -17367.073,E2 -17367.073} C_VEL
LIN {X 0,Y 275.466,Z 391.894,A -85,B 0,C 180,E1 -17368.537,E2 -17368.537} C_VEL
LIN {X 0,Y 275.543,Z 392.421,A -85,B 0,C 180,E1 -17369.999,E2 -17369.999} C_VEL
LIN {X 0,Y 275.432,Z 392.503,A -85,B 0,C 180,E1 -17371.461,E2 -17371.461} C_VEL
LIN {X 0,Y 275.407,Z 392.169,A -85,B 0,C 180,E1 -17372.924,E2 -17372.924} C_VEL
LIN {X 0,Y 275.353,Z 390.323,A -85,B 0,C 180,E1 -17375.858,E2 -17375.858} C_VEL
LIN {X 0,Y 275.489,Z 388.779,A -85,B 0,C 180,E1 -17377.327,E2 -17377.327} C_VEL
LIN {X 0,Y 275.851,Z 385.657,A -85,B 0,C 180,E1 -17379.531,E2 -17379.531} C_VEL
LIN {X 0,Y 276.468,Z 381.496,A -85,B 0,C 180,E1 -17381.732,E2 -17381.732} C_VEL
LIN {X 0,Y 277.85,Z 375.176,A -85,B 0,C 180,E1 -17384.276,E2 -17384.276} C_VEL
LIN {X 0,Y 279.371,Z 368.35,A -85,B 0,C 180,E1 -17386.438,E2 -17386.438} C_VEL
LIN {X 0,Y 281.186,Z 359.976,A -85,B 0,C 180,E1 -17388.581,E2 -17388.581} C_VEL
LIN {X 0,Y 283.128,Z 351.445,A -85,B 0,C 180,E1 -17390.334,E2 -17390.334} C_VEL
LIN {X 0,Y 285.452,Z 341.014,A -85,B 0,C 180,E1 -17392.051,E2 -17392.051} C_VEL
LIN {X 0,Y 286.037,Z 333.671,A -85,B 0,C 180,E1 -17393.147,E2 -17393.147} C_VEL
LIN {X 0,Y 285.676,Z 321.895,A -85,B 0,C 180,E1 -17394.721,E2 -17394.721} C_VEL
LIN {X 0,Y 284.422,Z 310.182,A -85,B 0,C 180,E1 -17396.089,E2 -17396.089} C_VEL
LIN {X 0,Y 281.878,Z 297.338,A -85,B 0,C 180,E1 -17397.45,E2 -17397.45} C_VEL
LIN {X 0,Y 278.648,Z 286.404,A -85,B 0,C 180,E1 -17398.524,E2 -17398.524} C_VEL
LIN {X 0,Y 277.862,Z 283.15,A -85,B 0,C 180,E1 -17398.824,E2 -17398.824} C_VEL
LIN {X 0,Y 278.983,Z 277.664,A -85,B 0,C 180,E1 -17402.792,E2 -17402.792} C_VEL
LIN {X 0,Y 279.79,Z 274.342,A -85,B 0,C 180,E1 -17405.289,E2 -17405.289} C_VEL
LIN {X 0,Y 280.192,Z 272.142,A -85,B 0,C 180,E1 -17407.01,E2 -17407.01} C_VEL
LIN {X 0,Y 279.859,Z 268.908,A -85,B 0,C 180,E1 -17409.817,E2 -17409.817} C_VEL
LIN {X 0,Y 279.279,Z 265.397,A -85,B 0,C 180,E1 -17413.13,E2 -17413.13} C_VEL
LIN {X 0,Y 278.602,Z 261.634,A -85,B 0,C 180,E1 -17417.068,E2 -17417.068} C_VEL
LIN {X 0,Y 278.057,Z 258.467,A -85,B 0,C 180,E1 -17420.808,E2 -17420.808} C_VEL
LIN {X 0,Y 277.6,Z 255.818,A -85,B 0,C 180,E1 -17424.386,E2 -17424.386} C_VEL
LIN {X 0,Y 277.315,Z 254.287,A -85,B 0,C 180,E1 -17426.751,E2 -17426.751} C_VEL
LIN {X 0,Y 277.243,Z 253.954,A -85,B 0,C 180,E1 -17427.834,E2 -17427.834} C_VEL
LIN {X 0,Y 277.287,Z 253.947,A -85,B 0,C 180,E1 -17431.21,E2 -17431.21} C_VEL
LIN {X 0,Y 277.311,Z 253.943,A -85,B 0,C 180,E1 -17434.477,E2 -17434.477} C_VEL
LIN {X 0,Y 277.282,Z 253.946,A -85,B 0,C 180,E1 -17437.652,E2 -17437.652} C_VEL
LIN {X 0,Y 277.342,Z 253.939,A -85,B 0,C 180,E1 -17440.764,E2 -17440.764} C_VEL
LIN {X 0,Y 277.431,Z 253.928,A -85,B 0,C 180,E1 -17445.324,E2 -17445.324} C_VEL
LIN {X 0,Y 277.503,Z 253.919,A -85,B 0,C 180,E1 -17449.786,E2 -17449.786} C_VEL
LIN {X 0,Y 277.648,Z 253.901,A -85,B 0,C 180,E1 -17452.727,E2 -17452.727} C_VEL
LIN {X 0,Y 277.816,Z 253.88,A -85,B 0,C 180,E1 -17458.548,E2 -17458.548} C_VEL
LIN {X 0,Y 277.816,Z 253.881,A -85,B 0,C 180,E1 -17461.447,E2 -17461.447} C_VEL
LIN {X 0,Y 277.646,Z 253.899,A -85,B 0,C 180,E1 -17467.269,E2 -17467.269} C_VEL
LIN {X 0,Y 277.499,Z 253.919,A -85,B 0,C 180,E1 -17470.209,E2 -17470.209} C_VEL
LIN {X 0,Y 277.426,Z 253.928,A -85,B 0,C 180,E1 -17471.69,E2 -17471.69} C_VEL
LIN {X 0,Y 277.522,Z 255.097,A -85,B 0,C 180,E1 -17474.667,E2 -17474.667} C_VEL
LIN {X 0,Y 277.564,Z 256.706,A -85,B 0,C 180,E1 -17477.686,E2 -17477.686} C_VEL
LIN {X 0,Y 277.392,Z 258.483,A -85,B 0,C 180,E1 -17480.773,E2 -17480.773} C_VEL
LIN {X 0,Y 277.145,Z 260.664,A -85,B 0,C 180,E1 -17484.245,E2 -17484.245} C_VEL
LIN {X 0,Y 278.269,Z 263.796,A -85,B 0,C 180,E1 -17484.581,E2 -17484.581} C_VEL
LIN {X 0,Y 282.758,Z 274.102,A -85,B 0,C 180,E1 -17485.879,E2 -17485.879} C_VEL
LIN {X 0,Y 286.53,Z 285.582,A -85,B 0,C 180,E1 -17487.378,E2 -17487.378} C_VEL
LIN {X 0,Y 289.035,Z 296.605,A -85,B 0,C 180,E1 -17488.916,E2 -17488.916} C_VEL
LIN {X 0,Y 289.686,Z 301.422,A -85,B 0,C 180,E1 -17489.622,E2 -17489.622} C_VEL
LIN {X 0,Y 287.531,Z 313.097,A -85,B 0,C 180,E1 -17491.189,E2 -17491.189} C_VEL
LIN {X 0,Y 285.674,Z 322.407,A -85,B 0,C 180,E1 -17492.764,E2 -17492.764} C_VEL
LIN {X 0,Y 283.832,Z 330.546,A -85,B 0,C 180,E1 -17494.443,E2 -17494.443} C_VEL
LIN {X 0,Y 281.874,Z 338.515,A -85,B 0,C 180,E1 -17496.462,E2 -17496.462} C_VEL
LIN {X 0,Y 280.264,Z 344.699,A -85,B 0,C 180,E1 -17498.409,E2 -17498.409} C_VEL
LIN {X 0,Y 278.584,Z 351.078,A -85,B 0,C 180,E1 -17500.985,E2 -17500.985} C_VEL
LIN {X 0,Y 277.513,Z 355.133,A -85,B 0,C 180,E1 -17503.135,E2 -17503.135} C_VEL
LIN {X 0,Y 276.63,Z 358.229,A -85,B 0,C 180,E1 -17505.342,E2 -17505.342} C_VEL
LIN {X 0,Y 275.951,Z 360.379,A -85,B 0,C 180,E1 -17507.606,E2 -17507.606} C_VEL
LIN {X 0,Y 275.48,Z 361.69,A -85,B 0,C 180,E1 -17510.374,E2 -17510.374} C_VEL
LIN {X 0,Y 275.315,Z 361.747,A -85,B 0,C 180,E1 -17512.306,E2 -17512.306} C_VEL
LIN {X 0,Y 275.311,Z 360.835,A -85,B 0,C 180,E1 -17514.768,E2 -17514.768} C_VEL
LIN {X 0,Y 275.643,Z 358.364,A -85,B 0,C 180,E1 -17517.629,E2 -17517.629} C_VEL
LIN {X 0,Y 276.301,Z 354.132,A -85,B 0,C 180,E1 -17520.527,E2 -17520.527} C_VEL
LIN {X 0,Y 276.919,Z 349.485,A -85,B 0,C 180,E1 -17522.819,E2 -17522.819} C_VEL
LIN {X 0,Y 277.869,Z 343.651,A -85,B 0,C 180,E1 -17525.055,E2 -17525.055} C_VEL
LIN {X 0,Y 278.912,Z 337.286,A -85,B 0,C 180,E1 -17527.012,E2 -17527.012} C_VEL
LIN {X 0,Y 280.268,Z 328.826,A -85,B 0,C 180,E1 -17529.111,E2 -17529.111} C_VEL
LIN {X 0,Y 281.929,Z 318.832,A -85,B 0,C 180,E1 -17531.092,E2 -17531.092} C_VEL
LIN {X 0,Y 283.354,Z 308.865,A -85,B 0,C 180,E1 -17532.686,E2 -17532.686} C_VEL
LIN {X 0,Y 284.84,Z 296.882,A -85,B 0,C 180,E1 -17534.2,E2 -17534.2} C_VEL
LIN {X 0,Y 285.092,Z 294.626,A -85,B 0,C 180,E1 -17534.451,E2 -17534.451} C_VEL
LIN {X 0,Y 282.874,Z 282.715,A -85,B 0,C 180,E1 -17535.799,E2 -17535.799} C_VEL
LIN {X 0,Y 279.675,Z 269.656,A -85,B 0,C 180,E1 -17537.023,E2 -17537.023} C_VEL
LIN {X 0,Y 276.373,Z 257.771,A -85,B 0,C 180,E1 -17537.938,E2 -17537.938} C_VEL
LIN {X 0,Y 276.745,Z 254.018,A -85,B 0,C 180,E1 -17542.707,E2 -17542.707} C_VEL
LIN {X 0,Y 277.06,Z 253.975,A -85,B 0,C 180,E1 -17545.637,E2 -17545.637} C_VEL
LIN {X 0,Y 277.653,Z 253.897,A -85,B 0,C 180,E1 -17548.551,E2 -17548.551} C_VEL
LIN {X 0,Y 277.809,Z 253.882,A -85,B 0,C 180,E1 -17551.451,E2 -17551.451} C_VEL
LIN {X 0,Y 277.64,Z 253.902,A -85,B 0,C 180,E1 -17557.273,E2 -17557.273} C_VEL
LIN {X 0,Y 277.495,Z 253.916,A -85,B 0,C 180,E1 -17560.213,E2 -17560.213} C_VEL
LIN {X 0,Y 277.424,Z 253.925,A -85,B 0,C 180,E1 -17564.676,E2 -17564.676} C_VEL
LIN {X 0,Y 277.363,Z 253.937,A -85,B 0,C 180,E1 -17569.234,E2 -17569.234} C_VEL
LIN {X 0,Y 277.321,Z 253.939,A -85,B 0,C 180,E1 -17573.923,E2 -17573.923} C_VEL
LIN {X 0,Y 277.319,Z 253.94,A -85,B 0,C 180,E1 -17577.509,E2 -17577.509} C_VEL
LIN {X 0,Y 277.264,Z 253.949,A -85,B 0,C 180,E1 -17580.484,E2 -17580.484} C_VEL
LIN {X 0,Y 277.247,Z 253.947,A -85,B 0,C 180,E1 -17583.897,E2 -17583.897} C_VEL
LIN {X 0,Y 277.28,Z 253.944,A -85,B 0,C 180,E1 -17587.469,E2 -17587.469} C_VEL
LIN {X 0,Y 277.259,Z 253.947,A -85,B 0,C 180,E1 -17591.229,E2 -17591.229} C_VEL
LIN {X 0,Y 277.245,Z 253.947,A -85,B 0,C 180,E1 -17595.219,E2 -17595.219} C_VEL
LIN {X 0,Y 277.284,Z 253.943,A -85,B 0,C 180,E1 -17599.499,E2 -17599.499} C_VEL
LIN {X 0,Y 277.287,Z 253.942,A -85,B 0,C 180,E1 -17602.537,E2 -17602.537} C_VEL
LIN {X 0,Y 277.253,Z 253.941,A -85,B 0,C 180,E1 -17606.108,E2 -17606.108} C_VEL
LIN {X 0,Y 277.261,Z 253.944,A -85,B 0,C 180,E1 -17609.542,E2 -17609.542} C_VEL
LIN {X 0,Y 277.357,Z 253.934,A -85,B 0,C 180,E1 -17612.867,E2 -17612.867} C_VEL
LIN {X 0,Y 277.33,Z 253.939,A -85,B 0,C 180,E1 -17616.082,E2 -17616.082} C_VEL
LIN {X 0,Y 277.348,Z 253.929,A -85,B 0,C 180,E1 -17620.769,E2 -17620.769} C_VEL
LIN {X 0,Y 277.439,Z 253.923,A -85,B 0,C 180,E1 -17625.329,E2 -17625.329} C_VEL
LIN {X 0,Y 277.466,Z 253.923,A -85,B 0,C 180,E1 -17629.79,E2 -17629.79} C_VEL
LIN {X 0,Y 277.634,Z 253.894,A -85,B 0,C 180,E1 -17632.731,E2 -17632.731} C_VEL
LIN {X 0,Y 277.827,Z 253.874,A -85,B 0,C 180,E1 -17638.553,E2 -17638.553} C_VEL
LIN {X 0,Y 277.827,Z 253.878,A -85,B 0,C 180,E1 -17641.452,E2 -17641.452} C_VEL
LIN {X 0,Y 277.626,Z 253.897,A -85,B 0,C 180,E1 -17647.274,E2 -17647.274} C_VEL
LIN {X 0,Y 277.466,Z 253.919,A -85,B 0,C 180,E1 -17650.215,E2 -17650.215} C_VEL
LIN {X 0,Y 277.436,Z 253.927,A -85,B 0,C 180,E1 -17651.606,E2 -17651.606} C_VEL
LIN {X 0,Y 276.792,Z 254.014,A -85,B 0,C 180,E1 -17652.818,E2 -17652.818} C_VEL
LIN {X 0,Y 273.897,Z 254.369,A -85,B 0,C 180,E1 -17654.792,E2 -17654.792} C_VEL
LIN {X 0,Y 271.426,Z 254.671,A -85,B 0,C 180,E1 -17656.396,E2 -17656.396} C_VEL
LIN {X 0,Y 270.376,Z 254.802,A -85,B 0,C 180,E1 -17657.642,E2 -17657.642} C_VEL
LIN {X 0,Y 270.297,Z 254.808,A -85,B 0,C 180,E1 -17658.064,E2 -17658.064} C_VEL
LIN {X 0,Y 270.233,Z 254.824,A -85,B 0,C 180,E1 -17661.354,E2 -17661.354} C_VEL
LIN {X 0,Y 270.284,Z 254.815,A -85,B 0,C 180,E1 -17664.587,E2 -17664.587} C_VEL
LIN {X 0,Y 270.28,Z 254.813,A -85,B 0,C 180,E1 -17667.91,E2 -17667.91} C_VEL
LIN {X 0,Y 270.195,Z 254.83,A -85,B 0,C 180,E1 -17671.349,E2 -17671.349} C_VEL
LIN {X 0,Y 270.212,Z 254.826,A -85,B 0,C 180,E1 -17674.906,E2 -17674.906} C_VEL
LIN {X 0,Y 270.208,Z 254.826,A -85,B 0,C 180,E1 -17678.711,E2 -17678.711} C_VEL
LIN {X 0,Y 270.243,Z 254.961,A -85,B 0,C 180,E1 -17680.917,E2 -17680.917} C_VEL
LIN {X 0,Y 270.925,Z 258.907,A -85,B 0,C 180,E1 -17684.462,E2 -17684.462} C_VEL
LIN {X 0,Y 271.817,Z 263.761,A -85,B 0,C 180,E1 -17688.577,E2 -17688.577} C_VEL
LIN {X 0,Y 272.462,Z 267.708,A -85,B 0,C 180,E1 -17691.75,E2 -17691.75} C_VEL
LIN {X 0,Y 272.495,Z 270.15,A -85,B 0,C 180,E1 -17693.614,E2 -17693.614} C_VEL
LIN {X 0,Y 272.006,Z 273.121,A -85,B 0,C 180,E1 -17695.775,E2 -17695.775} C_VEL
LIN {X 0,Y 270.718,Z 279.662,A -85,B 0,C 180,E1 -17700.444,E2 -17700.444} C_VEL
LIN {X 0,Y 269.86,Z 285.649,A -85,B 0,C 180,E1 -17704.546,E2 -17704.546} C_VEL
LIN {X 0,Y 272.19,Z 299.273,A -85,B 0,C 180,E1 -17705.42,E2 -17705.42} C_VEL
LIN {X 0,Y 274.026,Z 312.856,A -85,B 0,C 180,E1 -17706.592,E2 -17706.592} C_VEL
LIN {X 0,Y 275.04,Z 324.656,A -85,B 0,C 180,E1 -17707.857,E2 -17707.857} C_VEL
LIN {X 0,Y 275.533,Z 335.5,A -85,B 0,C 180,E1 -17709.272,E2 -17709.272} C_VEL
LIN {X 0,Y 273.868,Z 346.249,A -85,B 0,C 180,E1 -17710.9,E2 -17710.9} C_VEL
LIN {X 0,Y 272.207,Z 356.733,A -85,B 0,C 180,E1 -17712.893,E2 -17712.893} C_VEL
LIN {X 0,Y 271.127,Z 363.951,A -85,B 0,C 180,E1 -17714.59,E2 -17714.59} C_VEL
LIN {X 0,Y 269.937,Z 371.756,A -85,B 0,C 180,E1 -17716.83,E2 -17716.83} C_VEL
LIN {X 0,Y 269.133,Z 377.069,A -85,B 0,C 180,E1 -17718.704,E2 -17718.704} C_VEL
LIN {X 0,Y 268.65,Z 382.229,A -85,B 0,C 180,E1 -17720.968,E2 -17720.968} C_VEL
LIN {X 0,Y 268.39,Z 386.208,A -85,B 0,C 180,E1 -17723.231,E2 -17723.231} C_VEL
LIN {X 0,Y 268.353,Z 389.121,A -85,B 0,C 180,E1 -17725.492,E2 -17725.492} C_VEL
LIN {X 0,Y 268.365,Z 390.482,A -85,B 0,C 180,E1 -17726.996,E2 -17726.996} C_VEL
LIN {X 0,Y 268.383,Z 391.431,A -85,B 0,C 180,E1 -17728.498,E2 -17728.498} C_VEL
LIN {X 0,Y 268.455,Z 391.981,A -85,B 0,C 180,E1 -17729.998,E2 -17729.998} C_VEL
LIN {X 0,Y 268.35,Z 392.109,A -85,B 0,C 180,E1 -17731.499,E2 -17731.499} C_VEL
LIN {X 0,Y 268.331,Z 391.802,A -85,B 0,C 180,E1 -17733.001,E2 -17733.001} C_VEL
LIN {X 0,Y 268.29,Z 390.001,A -85,B 0,C 180,E1 -17736.013,E2 -17736.013} C_VEL
LIN {X 0,Y 268.404,Z 388.5,A -85,B 0,C 180,E1 -17737.521,E2 -17737.521} C_VEL
LIN {X 0,Y 268.797,Z 385.417,A -85,B 0,C 180,E1 -17739.783,E2 -17739.783} C_VEL
LIN {X 0,Y 269.476,Z 381.305,A -85,B 0,C 180,E1 -17742.041,E2 -17742.041} C_VEL
LIN {X 0,Y 270.967,Z 375.085,A -85,B 0,C 180,E1 -17744.647,E2 -17744.647} C_VEL
LIN {X 0,Y 272.547,Z 368.419,A -85,B 0,C 180,E1 -17746.842,E2 -17746.842} C_VEL
LIN {X 0,Y 274.452,Z 360.071,A -85,B 0,C 180,E1 -17749.054,E2 -17749.054} C_VEL
LIN {X 0,Y 276.478,Z 351.664,A -85,B 0,C 180,E1 -17750.846,E2 -17750.846} C_VEL
LIN {X 0,Y 278.883,Z 341.394,A -85,B 0,C 180,E1 -17752.599,E2 -17752.599} C_VEL
LIN {X 0,Y 279.48,Z 332.739,A -85,B 0,C 180,E1 -17753.937,E2 -17753.937} C_VEL
LIN {X 0,Y 279.132,Z 320.739,A -85,B 0,C 180,E1 -17755.584,E2 -17755.584} C_VEL
LIN {X 0,Y 277.81,Z 309.818,A -85,B 0,C 180,E1 -17756.927,E2 -17756.927} C_VEL
LIN {X 0,Y 275.46,Z 298.25,A -85,B 0,C 180,E1 -17758.223,E2 -17758.223} C_VEL
LIN {X 0,Y 272.134,Z 286.513,A -85,B 0,C 180,E1 -17759.445,E2 -17759.445} C_VEL
LIN {X 0,Y 271.074,Z 283.199,A -85,B 0,C 180,E1 -17759.77,E2 -17759.77} C_VEL
LIN {X 0,Y 271.035,Z 282.65,A -85,B 0,C 180,E1 -17759.835,E2 -17759.835} C_VEL
LIN {X 0,Y 271.967,Z 278.622,A -85,B 0,C 180,E1 -17762.864,E2 -17762.864} C_VEL
LIN {X 0,Y 272.987,Z 274.215,A -85,B 0,C 180,E1 -17766.306,E2 -17766.306} C_VEL
LIN {X 0,Y 273.134,Z 272.05,A -85,B 0,C 180,E1 -17768.135,E2 -17768.135} C_VEL
LIN {X 0,Y 272.578,Z 268.31,A -85,B 0,C 180,E1 -17771.604,E2 -17771.604} C_VEL
LIN {X 0,Y 271.825,Z 264.317,A -85,B 0,C 180,E1 -17775.724,E2 -17775.724} C_VEL
LIN {X 0,Y 271.265,Z 260.944,A -85,B 0,C 180,E1 -17779.629,E2 -17779.629} C_VEL
LIN {X 0,Y 270.78,Z 257.989,A -85,B 0,C 180,E1 -17783.568,E2 -17783.568} C_VEL
LIN {X 0,Y 270.38,Z 255.831,A -85,B 0,C 180,E1 -17786.915,E2 -17786.915} C_VEL
LIN {X 0,Y 270.184,Z 254.843,A -85,B 0,C 180,E1 -17788.65,E2 -17788.65} C_VEL
LIN {X 0,Y 270.263,Z 254.821,A -85,B 0,C 180,E1 -17792.143,E2 -17792.143} C_VEL
LIN {X 0,Y 270.275,Z 254.82,A -85,B 0,C 180,E1 -17795.517,E2 -17795.517} C_VEL
LIN {X 0,Y 270.299,Z 254.815,A -85,B 0,C 180,E1 -17800.242,E2 -17800.242} C_VEL
LIN {X 0,Y 270.399,Z 254.804,A -85,B 0,C 180,E1 -17804.933,E2 -17804.933} C_VEL
LIN {X 0,Y 270.438,Z 254.8,A -85,B 0,C 180,E1 -17809.517,E2 -17809.517} C_VEL
LIN {X 0,Y 270.606,Z 254.779,A -85,B 0,C 180,E1 -17812.536,E2 -17812.536} C_VEL
LIN {X 0,Y 270.782,Z 254.756,A -85,B 0,C 180,E1 -17818.51,E2 -17818.51} C_VEL
LIN {X 0,Y 270.782,Z 254.757,A -85,B 0,C 180,E1 -17821.485,E2 -17821.485} C_VEL
LIN {X 0,Y 270.604,Z 254.777,A -85,B 0,C 180,E1 -17827.459,E2 -17827.459} C_VEL
LIN {X 0,Y 270.434,Z 254.798,A -85,B 0,C 180,E1 -17830.479,E2 -17830.479} C_VEL
LIN {X 0,Y 270.49,Z 255.851,A -85,B 0,C 180,E1 -17833.521,E2 -17833.521} C_VEL
LIN {X 0,Y 270.552,Z 257.374,A -85,B 0,C 180,E1 -17836.601,E2 -17836.601} C_VEL
LIN {X 0,Y 270.47,Z 259.093,A -85,B 0,C 180,E1 -17839.74,E2 -17839.74} C_VEL
LIN {X 0,Y 270.234,Z 261.312,A -85,B 0,C 180,E1 -17843.211,E2 -17843.211} C_VEL
LIN {X 0,Y 271.525,Z 264.573,A -85,B 0,C 180,E1 -17843.599,E2 -17843.599} C_VEL
LIN {X 0,Y 276.21,Z 275.24,A -85,B 0,C 180,E1 -17845.05,E2 -17845.05} C_VEL
LIN {X 0,Y 279.83,Z 286.095,A -85,B 0,C 180,E1 -17846.547,E2 -17846.547} C_VEL
LIN {X 0,Y 282.245,Z 296.23,A -85,B 0,C 180,E1 -17848.031,E2 -17848.031} C_VEL
LIN {X 0,Y 283.274,Z 302.94,A -85,B 0,C 180,E1 -17849.077,E2 -17849.077} C_VEL
LIN {X 0,Y 280.983,Z 314.613,A -85,B 0,C 180,E1 -17850.71,E2 -17850.71} C_VEL
LIN {X 0,Y 278.91,Z 324.294,A -85,B 0,C 180,E1 -17852.424,E2 -17852.424} C_VEL
LIN {X 0,Y 276.776,Z 333.165,A -85,B 0,C 180,E1 -17854.389,E2 -17854.389} C_VEL
LIN {X 0,Y 274.548,Z 341.316,A -85,B 0,C 180,E1 -17856.638,E2 -17856.638} C_VEL
LIN {X 0,Y 272.966,Z 347.228,A -85,B 0,C 180,E1 -17858.705,E2 -17858.705} C_VEL
LIN {X 0,Y 271.324,Z 353.024,A -85,B 0,C 180,E1 -17861.31,E2 -17861.31} C_VEL
LIN {X 0,Y 270.363,Z 356.403,A -85,B 0,C 180,E1 -17863.296,E2 -17863.296} C_VEL
LIN {X 0,Y 269.568,Z 358.909,A -85,B 0,C 180,E1 -17865.259,E2 -17865.259} C_VEL
LIN {X 0,Y 268.971,Z 360.691,A -85,B 0,C 180,E1 -17867.209,E2 -17867.209} C_VEL
LIN {X 0,Y 268.497,Z 361.881,A -85,B 0,C 180,E1 -17869.379,E2 -17869.379} C_VEL
LIN {X 0,Y 268.246,Z 362.21,A -85,B 0,C 180,E1 -17871.808,E2 -17871.808} C_VEL
LIN {X 0,Y 268.218,Z 361.461,A -85,B 0,C 180,E1 -17874.314,E2 -17874.314} C_VEL
LIN {X 0,Y 268.43,Z 359.512,A -85,B 0,C 180,E1 -17876.905,E2 -17876.905} C_VEL
LIN {X 0,Y 268.928,Z 356.193,A -85,B 0,C 180,E1 -17879.581,E2 -17879.581} C_VEL
LIN {X 0,Y 269.573,Z 351.917,A -85,B 0,C 180,E1 -17882.014,E2 -17882.014} C_VEL
LIN {X 0,Y 270.53,Z 345.936,A -85,B 0,C 180,E1 -17884.565,E2 -17884.565} C_VEL
LIN {X 0,Y 271.652,Z 339.343,A -85,B 0,C 180,E1 -17886.765,E2 -17886.765} C_VEL
LIN {X 0,Y 272.956,Z 331.507,A -85,B 0,C 180,E1 -17888.873,E2 -17888.873} C_VEL
LIN {X 0,Y 274.554,Z 322.135,A -85,B 0,C 180,E1 -17890.9,E2 -17890.9} C_VEL
LIN {X 0,Y 276.27,Z 311.028,A -85,B 0,C 180,E1 -17892.8,E2 -17892.8} C_VEL
LIN {X 0,Y 277.713,Z 300.11,A -85,B 0,C 180,E1 -17894.293,E2 -17894.293} C_VEL
LIN {X 0,Y 278.233,Z 295.636,A -85,B 0,C 180,E1 -17894.809,E2 -17894.809} C_VEL
LIN {X 0,Y 276.075,Z 283.938,A -85,B 0,C 180,E1 -17896.194,E2 -17896.194} C_VEL
LIN {X 0,Y 272.868,Z 270.581,A -85,B 0,C 180,E1 -17897.497,E2 -17897.497} C_VEL
LIN {X 0,Y 269.325,Z 258.163,A -85,B 0,C 180,E1 -17898.477,E2 -17898.477} C_VEL
LIN {X 0,Y 269.677,Z 255.01,A -85,B 0,C 180,E1 -17902.514,E2 -17902.514} C_VEL
LIN {X 0,Y 270.007,Z 254.853,A -85,B 0,C 180,E1 -17905.523,E2 -17905.523} C_VEL
LIN {X 0,Y 270.586,Z 254.777,A -85,B 0,C 180,E1 -17908.513,E2 -17908.513} C_VEL
LIN {X 0,Y 270.799,Z 254.751,A -85,B 0,C 180,E1 -17910.001,E2 -17910.001} C_VEL
LIN {X 0,Y 270.619,Z 254.776,A -85,B 0,C 180,E1 -17912.979,E2 -17912.979} C_VEL
LIN {X 0,Y 270.598,Z 254.778,A -85,B 0,C 180,E1 -17917.463,E2 -17917.463} C_VEL
LIN {X 0,Y 270.43,Z 254.797,A -85,B 0,C 180,E1 -17920.483,E2 -17920.483} C_VEL
LIN {X 0,Y 270.392,Z 254.803,A -85,B 0,C 180,E1 -17925.067,E2 -17925.067} C_VEL
LIN {X 0,Y 270.317,Z 254.812,A -85,B 0,C 180,E1 -17929.756,E2 -17929.756} C_VEL
LIN {X 0,Y 270.265,Z 254.82,A -85,B 0,C 180,E1 -17934.588,E2 -17934.588} C_VEL
LIN {X 0,Y 270.264,Z 254.819,A -85,B 0,C 180,E1 -17937.911,E2 -17937.911} C_VEL
LIN {X 0,Y 270.176,Z 254.831,A -85,B 0,C 180,E1 -17941.351,E2 -17941.351} C_VEL
LIN {X 0,Y 270.208,Z 254.829,A -85,B 0,C 180,E1 -17944.906,E2 -17944.906} C_VEL
LIN {X 0,Y 270.216,Z 254.826,A -85,B 0,C 180,E1 -17948.72,E2 -17948.72} C_VEL
LIN {X 0,Y 270.217,Z 254.828,A -85,B 0,C 180,E1 -17952.551,E2 -17952.551} C_VEL
LIN {X 0,Y 270.2,Z 254.828,A -85,B 0,C 180,E1 -17956.745,E2 -17956.745} C_VEL
LIN {X 0,Y 270.234,Z 254.821,A -85,B 0,C 180,E1 -17959.449,E2 -17959.449} C_VEL
LIN {X 0,Y 270.256,Z 254.814,A -85,B 0,C 180,E1 -17963.724,E2 -17963.724} C_VEL
LIN {X 0,Y 270.203,Z 254.821,A -85,B 0,C 180,E1 -17966.896,E2 -17966.896} C_VEL
LIN {X 0,Y 270.219,Z 254.826,A -85,B 0,C 180,E1 -17970.389,E2 -17970.389} C_VEL
LIN {X 0,Y 270.263,Z 254.819,A -85,B 0,C 180,E1 -17973.767,E2 -17973.767} C_VEL
LIN {X 0,Y 270.234,Z 254.817,A -85,B 0,C 180,E1 -17977.042,E2 -17977.042} C_VEL
LIN {X 0,Y 270.304,Z 254.807,A -85,B 0,C 180,E1 -17980.247,E2 -17980.247} C_VEL
LIN {X 0,Y 270.407,Z 254.798,A -85,B 0,C 180,E1 -17984.938,E2 -17984.938} C_VEL
LIN {X 0,Y 270.418,Z 254.799,A -85,B 0,C 180,E1 -17989.521,E2 -17989.521} C_VEL
LIN {X 0,Y 270.591,Z 254.771,A -85,B 0,C 180,E1 -17992.541,E2 -17992.541} C_VEL
LIN {X 0,Y 270.793,Z 254.751,A -85,B 0,C 180,E1 -17998.515,E2 -17998.515} C_VEL
LIN {X 0,Y 270.793,Z 254.754,A -85,B 0,C 180,E1 -18001.489,E2 -18001.489} C_VEL
LIN {X 0,Y 270.584,Z 254.774,A -85,B 0,C 180,E1 -18007.464,E2 -18007.464} C_VEL
LIN {X 0,Y 270.419,Z 254.796,A -85,B 0,C 180,E1 -18010.484,E2 -18010.484} C_VEL
LIN {X 0,Y 270.413,Z 254.801,A -85,B 0,C 180,E1 -18015.066,E2 -18015.066} C_VEL
LIN {X 0,Y 270.297,Z 254.808,A -85,B 0,C 180,E1 -18018.064,E2 -18018.064} C_VEL
LIN {X 0,Y 269.629,Z 254.896,A -85,B 0,C 180,E1 -18019.306,E2 -18019.306} C_VEL
LIN {X 0,Y 266.721,Z 255.261,A -85,B 0,C 180,E1 -18021.33,E2 -18021.33} C_VEL
LIN {X 0,Y 264.28,Z 255.565,A -85,B 0,C 180,E1 -18022.975,E2 -18022.975} C_VEL
LIN {X 0,Y 263.281,Z 255.688,A -85,B 0,C 180,E1 -18024.253,E2 -18024.253} C_VEL
LIN {X 0,Y 263.227,Z 255.695,A -85,B 0,C 180,E1 -18024.685,E2 -18024.685} C_VEL
LIN {X 0,Y 263.176,Z 255.698,A -85,B 0,C 180,E1 -18028.732,E2 -18028.732} C_VEL
LIN {X 0,Y 263.143,Z 255.705,A -85,B 0,C 180,E1 -18032.289,E2 -18032.289} C_VEL
LIN {X 0,Y 263.192,Z 255.7,A -85,B 0,C 180,E1 -18036.764,E2 -18036.764} C_VEL
LIN {X 0,Y 263.237,Z 255.871,A -85,B 0,C 180,E1 -18040.602,E2 -18040.602} C_VEL
LIN {X 0,Y 263.998,Z 260.53,A -85,B 0,C 180,E1 -18044.877,E2 -18044.877} C_VEL
LIN {X 0,Y 264.779,Z 264.623,A -85,B 0,C 180,E1 -18048.425,E2 -18048.425} C_VEL
LIN {X 0,Y 265.374,Z 268.335,A -85,B 0,C 180,E1 -18051.51,E2 -18051.51} C_VEL
LIN {X 0,Y 265.456,Z 270.848,A -85,B 0,C 180,E1 -18053.479,E2 -18053.479} C_VEL
LIN {X 0,Y 264.81,Z 274.376,A -85,B 0,C 180,E1 -18056.127,E2 -18056.127} C_VEL
LIN {X 0,Y 263.623,Z 280.284,A -85,B 0,C 180,E1 -18060.447,E2 -18060.447} C_VEL
LIN {X 0,Y 262.872,Z 285.202,A -85,B 0,C 180,E1 -18063.966,E2 -18063.966} C_VEL
LIN {X 0,Y 265.199,Z 298.748,A -85,B 0,C 180,E1 -18064.858,E2 -18064.858} C_VEL
LIN {X 0,Y 267.033,Z 312.233,A -85,B 0,C 180,E1 -18066.057,E2 -18066.057} C_VEL
LIN {X 0,Y 268.056,Z 323.852,A -85,B 0,C 180,E1 -18067.336,E2 -18067.336} C_VEL
LIN {X 0,Y 268.538,Z 334.172,A -85,B 0,C 180,E1 -18068.706,E2 -18068.706} C_VEL
LIN {X 0,Y 268.073,Z 339.42,A -85,B 0,C 180,E1 -18069.471,E2 -18069.471} C_VEL
LIN {X 0,Y 266.398,Z 349.352,A -85,B 0,C 180,E1 -18071.143,E2 -18071.143} C_VEL
LIN {X 0,Y 264.921,Z 358.405,A -85,B 0,C 180,E1 -18073.032,E2 -18073.032} C_VEL
LIN {X 0,Y 263.717,Z 365.892,A -85,B 0,C 180,E1 -18074.938,E2 -18074.938} C_VEL
LIN {X 0,Y 262.571,Z 373.243,A -85,B 0,C 180,E1 -18077.241,E2 -18077.241} C_VEL
LIN {X 0,Y 261.918,Z 378.219,A -85,B 0,C 180,E1 -18079.172,E2 -18079.172} C_VEL
LIN {X 0,Y 261.487,Z 383.039,A -85,B 0,C 180,E1 -18081.498,E2 -18081.498} C_VEL
LIN {X 0,Y 261.298,Z 386.709,A -85,B 0,C 180,E1 -18083.822,E2 -18083.822} C_VEL
LIN {X 0,Y 261.262,Z 388.589,A -85,B 0,C 180,E1 -18085.37,E2 -18085.37} C_VEL
LIN {X 0,Y 261.294,Z 389.995,A -85,B 0,C 180,E1 -18086.915,E2 -18086.915} C_VEL
LIN {X 0,Y 261.303,Z 390.968,A -85,B 0,C 180,E1 -18088.457,E2 -18088.457} C_VEL
LIN {X 0,Y 261.369,Z 391.541,A -85,B 0,C 180,E1 -18089.998,E2 -18089.998} C_VEL
LIN {X 0,Y 261.271,Z 391.705,A -85,B 0,C 180,E1 -18091.54,E2 -18091.54} C_VEL
LIN {X 0,Y 261.234,Z 391.434,A -85,B 0,C 180,E1 -18093.083,E2 -18093.083} C_VEL
LIN {X 0,Y 261.222,Z 389.679,A -85,B 0,C 180,E1 -18096.176,E2 -18096.176} C_VEL
LIN {X 0,Y 261.336,Z 388.214,A -85,B 0,C 180,E1 -18097.726,E2 -18097.726} C_VEL
LIN {X 0,Y 261.751,Z 385.183,A -85,B 0,C 180,E1 -18100.049,E2 -18100.049} C_VEL
LIN {X 0,Y 262.498,Z 381.141,A -85,B 0,C 180,E1 -18102.366,E2 -18102.366} C_VEL
LIN {X 0,Y 264.094,Z 375.021,A -85,B 0,C 180,E1 -18105.037,E2 -18105.037} C_VEL
LIN {X 0,Y 266.002,Z 367.524,A -85,B 0,C 180,E1 -18107.557,E2 -18107.557} C_VEL
LIN {X 0,Y 268.118,Z 358.646,A -85,B 0,C 180,E1 -18109.922,E2 -18109.922} C_VEL
LIN {X 0,Y 270.796,Z 348.074,A -85,B 0,C 180,E1 -18112.104,E2 -18112.104} C_VEL
LIN {X 0,Y 272.546,Z 340.67,A -85,B 0,C 180,E1 -18113.356,E2 -18113.356} C_VEL
LIN {X 0,Y 272.964,Z 330.82,A -85,B 0,C 180,E1 -18114.932,E2 -18114.932} C_VEL
LIN {X 0,Y 272.515,Z 319.59,A -85,B 0,C 180,E1 -18116.516,E2 -18116.516} C_VEL
LIN {X 0,Y 270.989,Z 307.788,A -85,B 0,C 180,E1 -18118.011,E2 -18118.011} C_VEL
LIN {X 0,Y 268.082,Z 294.99,A -85,B 0,C 180,E1 -18119.523,E2 -18119.523} C_VEL
LIN {X 0,Y 264.792,Z 284.621,A -85,B 0,C 180,E1 -18120.686,E2 -18120.686} C_VEL
LIN {X 0,Y 264.295,Z 282.179,A -85,B 0,C 180,E1 -18120.928,E2 -18120.928} C_VEL
LIN {X 0,Y 265.515,Z 277.174,A -85,B 0,C 180,E1 -18124.857,E2 -18124.857} C_VEL
LIN {X 0,Y 266.164,Z 274.109,A -85,B 0,C 180,E1 -18127.393,E2 -18127.393} C_VEL
LIN {X 0,Y 265.886,Z 271.311,A -85,B 0,C 180,E1 -18129.953,E2 -18129.953} C_VEL
LIN {X 0,Y 265.267,Z 267.749,A -85,B 0,C 180,E1 -18133.537,E2 -18133.537} C_VEL
LIN {X 0,Y 264.518,Z 263.477,A -85,B 0,C 180,E1 -18138.375,E2 -18138.375} C_VEL
LIN {X 0,Y 263.994,Z 260.495,A -85,B 0,C 180,E1 -18142.241,E2 -18142.241} C_VEL
LIN {X 0,Y 263.567,Z 258.05,A -85,B 0,C 180,E1 -18145.944,E2 -18145.944} C_VEL
LIN {X 0,Y 263.223,Z 256.047,A -85,B 0,C 180,E1 -18149.514,E2 -18149.514} C_VEL
LIN {X 0,Y 263.191,Z 255.702,A -85,B 0,C 180,E1 -18153,E2 -18153} C_VEL
LIN {X 0,Y 263.182,Z 255.703,A -85,B 0,C 180,E1 -18156.385,E2 -18156.385} C_VEL
LIN {X 0,Y 263.261,Z 255.693,A -85,B 0,C 180,E1 -18159.691,E2 -18159.691} C_VEL
LIN {X 0,Y 263.347,Z 255.681,A -85,B 0,C 180,E1 -18164.52,E2 -18164.52} C_VEL
LIN {X 0,Y 263.37,Z 255.68,A -85,B 0,C 180,E1 -18169.232,E2 -18169.232} C_VEL
LIN {X 0,Y 263.568,Z 255.656,A -85,B 0,C 180,E1 -18172.336,E2 -18172.336} C_VEL
LIN {X 0,Y 263.746,Z 255.632,A -85,B 0,C 180,E1 -18178.471,E2 -18178.471} C_VEL
LIN {X 0,Y 263.746,Z 255.633,A -85,B 0,C 180,E1 -18181.525,E2 -18181.525} C_VEL
LIN {X 0,Y 263.565,Z 255.655,A -85,B 0,C 180,E1 -18187.659,E2 -18187.659} C_VEL
LIN {X 0,Y 263.535,Z 255.659,A -85,B 0,C 180,E1 -18189.357,E2 -18189.357} C_VEL
LIN {X 0,Y 263.466,Z 256.64,A -85,B 0,C 180,E1 -18192.319,E2 -18192.319} C_VEL
LIN {X 0,Y 263.579,Z 258.507,A -85,B 0,C 180,E1 -18196.288,E2 -18196.288} C_VEL
LIN {X 0,Y 263.424,Z 260.62,A -85,B 0,C 180,E1 -18200.291,E2 -18200.291} C_VEL
LIN {X 0,Y 263.263,Z 261.64,A -85,B 0,C 180,E1 -18202.047,E2 -18202.047} C_VEL
LIN {X 0,Y 264.57,Z 265.013,A -85,B 0,C 180,E1 -18202.497,E2 -18202.497} C_VEL
LIN {X 0,Y 268.897,Z 274.451,A -85,B 0,C 180,E1 -18203.868,E2 -18203.868} C_VEL
LIN {X 0,Y 272.633,Z 284.785,A -85,B 0,C 180,E1 -18205.395,E2 -18205.395} C_VEL
LIN {X 0,Y 275.236,Z 294.699,A -85,B 0,C 180,E1 -18206.908,E2 -18206.908} C_VEL
LIN {X 0,Y 276.851,Z 304.022,A -85,B 0,C 180,E1 -18208.42,E2 -18208.42} C_VEL
LIN {X 0,Y 274.677,Z 315.246,A -85,B 0,C 180,E1 -18210.052,E2 -18210.052} C_VEL
LIN {X 0,Y 272.597,Z 324.391,A -85,B 0,C 180,E1 -18211.705,E2 -18211.705} C_VEL
LIN {X 0,Y 270.329,Z 333.287,A -85,B 0,C 180,E1 -18213.705,E2 -18213.705} C_VEL
LIN {X 0,Y 267.897,Z 341.853,A -85,B 0,C 180,E1 -18216.124,E2 -18216.124} C_VEL
LIN {X 0,Y 265.898,Z 348.769,A -85,B 0,C 180,E1 -18218.661,E2 -18218.661} C_VEL
LIN {X 0,Y 264.537,Z 353.3,A -85,B 0,C 180,E1 -18220.789,E2 -18220.789} C_VEL
LIN {X 0,Y 263.486,Z 356.698,A -85,B 0,C 180,E1 -18222.821,E2 -18222.821} C_VEL
LIN {X 0,Y 262.948,Z 358.311,A -85,B 0,C 180,E1 -18224.017,E2 -18224.017} C_VEL
LIN {X 0,Y 262.114,Z 360.708,A -85,B 0,C 180,E1 -18226.377,E2 -18226.377} C_VEL
LIN {X 0,Y 261.548,Z 362.156,A -85,B 0,C 180,E1 -18228.793,E2 -18228.793} C_VEL
LIN {X 0,Y 261.159,Z 362.603,A -85,B 0,C 180,E1 -18231.763,E2 -18231.763} C_VEL
LIN {X 0,Y 261.124,Z 362.062,A -85,B 0,C 180,E1 -18233.841,E2 -18233.841} C_VEL
LIN {X 0,Y 261.283,Z 360.31,A -85,B 0,C 180,E1 -18236.49,E2 -18236.49} C_VEL
LIN {X 0,Y 261.798,Z 357.027,A -85,B 0,C 180,E1 -18239.334,E2 -18239.334} C_VEL
LIN {X 0,Y 262.488,Z 352.447,A -85,B 0,C 180,E1 -18242.068,E2 -18242.068} C_VEL
LIN {X 0,Y 263.3,Z 347.505,A -85,B 0,C 180,E1 -18244.296,E2 -18244.296} C_VEL
LIN {X 0,Y 264.407,Z 341.37,A -85,B 0,C 180,E1 -18246.505,E2 -18246.505} C_VEL
LIN {X 0,Y 265.704,Z 333.875,A -85,B 0,C 180,E1 -18248.674,E2 -18248.674} C_VEL
LIN {X 0,Y 267.324,Z 324.39,A -85,B 0,C 180,E1 -18250.871,E2 -18250.871} C_VEL
LIN {X 0,Y 268.967,Z 314.492,A -85,B 0,C 180,E1 -18252.711,E2 -18252.711} C_VEL
LIN {X 0,Y 270.554,Z 303.544,A -85,B 0,C 180,E1 -18254.33,E2 -18254.33} C_VEL
LIN {X 0,Y 271.373,Z 296.646,A -85,B 0,C 180,E1 -18255.184,E2 -18255.184} C_VEL
LIN {X 0,Y 269.189,Z 284.645,A -85,B 0,C 180,E1 -18256.664,E2 -18256.664} C_VEL
LIN {X 0,Y 266.039,Z 271.455,A -85,B 0,C 180,E1 -18257.992,E2 -18257.992} C_VEL
LIN {X 0,Y 262.304,Z 258.554,A -85,B 0,C 180,E1 -18259.045,E2 -18259.045} C_VEL
LIN {X 0,Y 262.599,Z 256.047,A -85,B 0,C 180,E1 -18262.311,E2 -18262.311} C_VEL
LIN {X 0,Y 262.826,Z 255.747,A -85,B 0,C 180,E1 -18263.861,E2 -18263.861} C_VEL
LIN {X 0,Y 263.522,Z 255.657,A -85,B 0,C 180,E1 -18268.473,E2 -18268.473} C_VEL
LIN {X 0,Y 263.758,Z 255.628,A -85,B 0,C 180,E1 -18270.002,E2 -18270.002} C_VEL
LIN {X 0,Y 263.553,Z 255.657,A -85,B 0,C 180,E1 -18273.059,E2 -18273.059} C_VEL
LIN {X 0,Y 263.56,Z 255.653,A -85,B 0,C 180,E1 -18277.664,E2 -18277.664} C_VEL
LIN {X 0,Y 263.363,Z 255.678,A -85,B 0,C 180,E1 -18280.768,E2 -18280.768} C_VEL
LIN {X 0,Y 263.34,Z 255.682,A -85,B 0,C 180,E1 -18285.48,E2 -18285.48} C_VEL
LIN {X 0,Y 263.278,Z 255.689,A -85,B 0,C 180,E1 -18290.307,E2 -18290.307} C_VEL
LIN {X 0,Y 263.2,Z 255.702,A -85,B 0,C 180,E1 -18295.294,E2 -18295.294} C_VEL
LIN {X 0,Y 263.172,Z 255.706,A -85,B 0,C 180,E1 -18298.732,E2 -18298.732} C_VEL
LIN {X 0,Y 263.126,Z 255.709,A -85,B 0,C 180,E1 -18302.291,E2 -18302.291} C_VEL
LIN {X 0,Y 263.182,Z 255.701,A -85,B 0,C 180,E1 -18305.981,E2 -18305.981} C_VEL
LIN {X 0,Y 263.154,Z 255.702,A -85,B 0,C 180,E1 -18309.866,E2 -18309.866} C_VEL
LIN {X 0,Y 263.141,Z 255.705,A -85,B 0,C 180,E1 -18313.982,E2 -18313.982} C_VEL
LIN {X 0,Y 263.147,Z 255.708,A -85,B 0,C 180,E1 -18318.403,E2 -18318.403} C_VEL
LIN {X 0,Y 263.186,Z 255.699,A -85,B 0,C 180,E1 -18322.111,E2 -18322.111} C_VEL
LIN {X 0,Y 263.183,Z 255.69,A -85,B 0,C 180,E1 -18325.894,E2 -18325.894} C_VEL
LIN {X 0,Y 263.147,Z 255.702,A -85,B 0,C 180,E1 -18329.51,E2 -18329.51} C_VEL
LIN {X 0,Y 263.192,Z 255.698,A -85,B 0,C 180,E1 -18333.006,E2 -18333.006} C_VEL
LIN {X 0,Y 263.186,Z 255.697,A -85,B 0,C 180,E1 -18336.39,E2 -18336.39} C_VEL
LIN {X 0,Y 263.266,Z 255.681,A -85,B 0,C 180,E1 -18339.696,E2 -18339.696} C_VEL
LIN {X 0,Y 263.355,Z 255.678,A -85,B 0,C 180,E1 -18344.525,E2 -18344.525} C_VEL
LIN {X 0,Y 263.36,Z 255.677,A -85,B 0,C 180,E1 -18349.236,E2 -18349.236} C_VEL
LIN {X 0,Y 263.55,Z 255.648,A -85,B 0,C 180,E1 -18352.34,E2 -18352.34} C_VEL
LIN {X 0,Y 263.757,Z 255.627,A -85,B 0,C 180,E1 -18358.476,E2 -18358.476} C_VEL
LIN {X 0,Y 263.757,Z 255.631,A -85,B 0,C 180,E1 -18361.529,E2 -18361.529} C_VEL
LIN {X 0,Y 263.546,Z 255.65,A -85,B 0,C 180,E1 -18367.665,E2 -18367.665} C_VEL
LIN {X 0,Y 263.359,Z 255.676,A -85,B 0,C 180,E1 -18370.768,E2 -18370.768} C_VEL
LIN {X 0,Y 263.361,Z 255.681,A -85,B 0,C 180,E1 -18375.48,E2 -18375.48} C_VEL
LIN {X 0,Y 263.274,Z 255.686,A -85,B 0,C 180,E1 -18380.308,E2 -18380.308} C_VEL
LIN {X 0,Y 263.227,Z 255.695,A -85,B 0,C 180,E1 -18384.685,E2 -18384.685} C_VEL
LIN {X 0,Y 262.627,Z 255.775,A -85,B 0,C 180,E1 -18385.962,E2 -18385.962} C_VEL
LIN {X 0,Y 259.775,Z 256.136,A -85,B 0,C 180,E1 -18388.042,E2 -18388.042} C_VEL
LIN {X 0,Y 257.292,Z 256.444,A -85,B 0,C 180,E1 -18389.734,E2 -18389.734} C_VEL
LIN {X 0,Y 256.2,Z 256.575,A -85,B 0,C 180,E1 -18391.047,E2 -18391.047} C_VEL
LIN {X 0,Y 256.1,Z 256.584,A -85,B 0,C 180,E1 -18391.493,E2 -18391.493} C_VEL
LIN {X 0,Y 256.092,Z 256.586,A -85,B 0,C 180,E1 -18395.194,E2 -18395.194} C_VEL
LIN {X 0,Y 256.096,Z 256.586,A -85,B 0,C 180,E1 -18399.14,E2 -18399.14} C_VEL
LIN {X 0,Y 256.155,Z 256.737,A -85,B 0,C 180,E1 -18400.221,E2 -18400.221} C_VEL
LIN {X 0,Y 256.96,Z 261.441,A -85,B 0,C 180,E1 -18404.672,E2 -18404.672} C_VEL
LIN {X 0,Y 257.901,Z 266.472,A -85,B 0,C 180,E1 -18409.153,E2 -18409.153} C_VEL
LIN {X 0,Y 258.387,Z 269.952,A -85,B 0,C 180,E1 -18412.075,E2 -18412.075} C_VEL
LIN {X 0,Y 258.408,Z 271.412,A -85,B 0,C 180,E1 -18413.247,E2 -18413.247} C_VEL
LIN {X 0,Y 257.766,Z 274.999,A -85,B 0,C 180,E1 -18416.016,E2 -18416.016} C_VEL
LIN {X 0,Y 256.34,Z 282.056,A -85,B 0,C 180,E1 -18421.326,E2 -18421.326} C_VEL
LIN {X 0,Y 255.898,Z 284.877,A -85,B 0,C 180,E1 -18423.374,E2 -18423.374} C_VEL
LIN {X 0,Y 258.266,Z 298.407,A -85,B 0,C 180,E1 -18424.302,E2 -18424.302} C_VEL
LIN {X 0,Y 260.03,Z 311.43,A -85,B 0,C 180,E1 -18425.485,E2 -18425.485} C_VEL
LIN {X 0,Y 261.079,Z 322.983,A -85,B 0,C 180,E1 -18426.783,E2 -18426.783} C_VEL
LIN {X 0,Y 261.602,Z 334.271,A -85,B 0,C 180,E1 -18428.32,E2 -18428.32} C_VEL
LIN {X 0,Y 261.437,Z 338.223,A -85,B 0,C 180,E1 -18428.926,E2 -18428.926} C_VEL
LIN {X 0,Y 259.618,Z 348.331,A -85,B 0,C 180,E1 -18430.632,E2 -18430.632} C_VEL
LIN {X 0,Y 258.042,Z 357.482,A -85,B 0,C 180,E1 -18432.565,E2 -18432.565} C_VEL
LIN {X 0,Y 256.823,Z 365.062,A -85,B 0,C 180,E1 -18434.524,E2 -18434.524} C_VEL
LIN {X 0,Y 255.616,Z 372.49,A -85,B 0,C 180,E1 -18436.888,E2 -18436.888} C_VEL
LIN {X 0,Y 254.7,Z 379.309,A -85,B 0,C 180,E1 -18439.666,E2 -18439.666} C_VEL
LIN {X 0,Y 254.317,Z 383.789,A -85,B 0,C 180,E1 -18442.056,E2 -18442.056} C_VEL
LIN {X 0,Y 254.236,Z 387.091,A -85,B 0,C 180,E1 -18444.383,E2 -18444.383} C_VEL
LIN {X 0,Y 254.224,Z 389.507,A -85,B 0,C 180,E1 -18446.829,E2 -18446.829} C_VEL
LIN {X 0,Y 254.225,Z 390.503,A -85,B 0,C 180,E1 -18448.414,E2 -18448.414} C_VEL
LIN {X 0,Y 254.285,Z 391.1,A -85,B 0,C 180,E1 -18449.998,E2 -18449.998} C_VEL
LIN {X 0,Y 254.193,Z 391.29,A -85,B 0,C 180,E1 -18451.583,E2 -18451.583} C_VEL
LIN {X 0,Y 254.14,Z 391.068,A -85,B 0,C 180,E1 -18453.169,E2 -18453.169} C_VEL
LIN {X 0,Y 254.152,Z 389.371,A -85,B 0,C 180,E1 -18456.349,E2 -18456.349} C_VEL
LIN {X 0,Y 254.266,Z 387.932,A -85,B 0,C 180,E1 -18457.942,E2 -18457.942} C_VEL
LIN {X 0,Y 254.726,Z 384.959,A -85,B 0,C 180,E1 -18460.33,E2 -18460.33} C_VEL
LIN {X 0,Y 255.529,Z 380.977,A -85,B 0,C 180,E1 -18462.709,E2 -18462.709} C_VEL
LIN {X 0,Y 256.936,Z 375.898,A -85,B 0,C 180,E1 -18465.06,E2 -18465.06} C_VEL
LIN {X 0,Y 258.648,Z 369.581,A -85,B 0,C 180,E1 -18467.389,E2 -18467.389} C_VEL
LIN {X 0,Y 260.682,Z 361.798,A -85,B 0,C 180,E1 -18469.693,E2 -18469.693} C_VEL
LIN {X 0,Y 263.281,Z 352.145,A -85,B 0,C 180,E1 -18471.943,E2 -18471.943} C_VEL
LIN {X 0,Y 265.862,Z 342.274,A -85,B 0,C 180,E1 -18473.772,E2 -18473.772} C_VEL
LIN {X 0,Y 266.478,Z 332.867,A -85,B 0,C 180,E1 -18475.367,E2 -18475.367} C_VEL
LIN {X 0,Y 266.22,Z 321.536,A -85,B 0,C 180,E1 -18477.069,E2 -18477.069} C_VEL
LIN {X 0,Y 264.886,Z 309.886,A -85,B 0,C 180,E1 -18478.654,E2 -18478.654} C_VEL
LIN {X 0,Y 262.327,Z 297.743,A -85,B 0,C 180,E1 -18480.188,E2 -18480.188} C_VEL
LIN {X 0,Y 258.57,Z 285.278,A -85,B 0,C 180,E1 -18481.69,E2 -18481.69} C_VEL
LIN {X 0,Y 257.614,Z 281.643,A -85,B 0,C 180,E1 -18482.119,E2 -18482.119} C_VEL
LIN {X 0,Y 258.679,Z 277.63,A -85,B 0,C 180,E1 -18485.403,E2 -18485.403} C_VEL
LIN {X 0,Y 259.023,Z 276.165,A -85,B 0,C 180,E1 -18486.648,E2 -18486.648} C_VEL
LIN {X 0,Y 259.043,Z 274.007,A -85,B 0,C 180,E1 -18488.607,E2 -18488.607} C_VEL
LIN {X 0,Y 258.637,Z 270.861,A -85,B 0,C 180,E1 -18491.702,E2 -18491.702} C_VEL
LIN {X 0,Y 258.016,Z 267.737,A -85,B 0,C 180,E1 -18495.086,E2 -18495.086} C_VEL
LIN {X 0,Y 257.448,Z 264.42,A -85,B 0,C 180,E1 -18499.065,E2 -18499.065} C_VEL
LIN {X 0,Y 256.991,Z 261.545,A -85,B 0,C 180,E1 -18503.01,E2 -18503.01} C_VEL
LIN {X 0,Y 256.546,Z 259.19,A -85,B 0,C 180,E1 -18506.775,E2 -18506.775} C_VEL
LIN {X 0,Y 256.211,Z 257.28,A -85,B 0,C 180,E1 -18510.41,E2 -18510.41} C_VEL
LIN {X 0,Y 256.14,Z 256.58,A -85,B 0,C 180,E1 -18512.194,E2 -18512.194} C_VEL
LIN {X 0,Y 256.165,Z 256.577,A -85,B 0,C 180,E1 -18515.697,E2 -18515.697} C_VEL
LIN {X 0,Y 256.164,Z 256.576,A -85,B 0,C 180,E1 -18519.102,E2 -18519.102} C_VEL
LIN {X 0,Y 256.296,Z 256.559,A -85,B 0,C 180,E1 -18524.083,E2 -18524.083} C_VEL
LIN {X 0,Y 256.306,Z 256.559,A -85,B 0,C 180,E1 -18528.932,E2 -18528.932} C_VEL
LIN {X 0,Y 256.535,Z 256.531,A -85,B 0,C 180,E1 -18532.125,E2 -18532.125} C_VEL
LIN {X 0,Y 256.709,Z 256.509,A -85,B 0,C 180,E1 -18538.429,E2 -18538.429} C_VEL
LIN {X 0,Y 256.709,Z 256.51,A -85,B 0,C 180,E1 -18541.566,E2 -18541.566} C_VEL
LIN {X 0,Y 256.532,Z 256.532,A -85,B 0,C 180,E1 -18547.871,E2 -18547.871} C_VEL
LIN {X 0,Y 256.518,Z 256.85,A -85,B 0,C 180,E1 -18549.499,E2 -18549.499} C_VEL
LIN {X 0,Y 256.561,Z 258.861,A -85,B 0,C 180,E1 -18554.27,E2 -18554.27} C_VEL
LIN {X 0,Y 256.556,Z 260.418,A -85,B 0,C 180,E1 -18557.535,E2 -18557.535} C_VEL
LIN {X 0,Y 256.398,Z 262.139,A -85,B 0,C 180,E1 -18560.82,E2 -18560.82} C_VEL
LIN {X 0,Y 257.523,Z 265.297,A -85,B 0,C 180,E1 -18561.256,E2 -18561.256} C_VEL
LIN {X 0,Y 258.764,Z 267.562,A -85,B 0,C 180,E1 -18561.626,E2 -18561.626} C_VEL
LIN {X 0,Y 263.176,Z 277.463,A -85,B 0,C 180,E1 -18563.194,E2 -18563.194} C_VEL
LIN {X 0,Y 266.609,Z 287.23,A -85,B 0,C 180,E1 -18564.735,E2 -18564.735} C_VEL
LIN {X 0,Y 269.304,Z 298.174,A -85,B 0,C 180,E1 -18566.522,E2 -18566.522} C_VEL
LIN {X 0,Y 270.48,Z 306.42,A -85,B 0,C 180,E1 -18567.944,E2 -18567.944} C_VEL
LIN {X 0,Y 268.31,Z 316.342,A -85,B 0,C 180,E1 -18569.437,E2 -18569.437} C_VEL
LIN {X 0,Y 265.711,Z 326.929,A -85,B 0,C 180,E1 -18571.463,E2 -18571.463} C_VEL
LIN {X 0,Y 263.395,Z 335.449,A -85,B 0,C 180,E1 -18573.509,E2 -18573.509} C_VEL
LIN {X 0,Y 261.3,Z 342.344,A -85,B 0,C 180,E1 -18575.553,E2 -18575.553} C_VEL
LIN {X 0,Y 259.473,Z 348.194,A -85,B 0,C 180,E1 -18577.708,E2 -18577.708} C_VEL
LIN {X 0,Y 257.775,Z 353.574,A -85,B 0,C 180,E1 -18580.238,E2 -18580.238} C_VEL
LIN {X 0,Y 256.628,Z 356.988,A -85,B 0,C 180,E1 -18582.32,E2 -18582.32} C_VEL
LIN {X 0,Y 255.696,Z 359.564,A -85,B 0,C 180,E1 -18584.39,E2 -18584.39} C_VEL
LIN {X 0,Y 254.998,Z 361.414,A -85,B 0,C 180,E1 -18586.449,E2 -18586.449} C_VEL
LIN {X 0,Y 254.517,Z 362.55,A -85,B 0,C 180,E1 -18588.495,E2 -18588.495} C_VEL
LIN {X 0,Y 254.181,Z 363.024,A -85,B 0,C 180,E1 -18590.727,E2 -18590.727} C_VEL
LIN {X 0,Y 254.018,Z 362.6,A -85,B 0,C 180,E1 -18593.35,E2 -18593.35} C_VEL
LIN {X 0,Y 254.204,Z 360.726,A -85,B 0,C 180,E1 -18596.433,E2 -18596.433} C_VEL
LIN {X 0,Y 254.765,Z 357.186,A -85,B 0,C 180,E1 -18599.549,E2 -18599.549} C_VEL
LIN {X 0,Y 255.4,Z 352.984,A -85,B 0,C 180,E1 -18602.11,E2 -18602.11} C_VEL
LIN {X 0,Y 256.383,Z 347.208,A -85,B 0,C 180,E1 -18604.762,E2 -18604.762} C_VEL
LIN {X 0,Y 257.618,Z 340.573,A -85,B 0,C 180,E1 -18607.125,E2 -18607.125} C_VEL
LIN {X 0,Y 258.994,Z 332.825,A -85,B 0,C 180,E1 -18609.345,E2 -18609.345} C_VEL
LIN {X 0,Y 260.718,Z 323.311,A -85,B 0,C 180,E1 -18611.536,E2 -18611.536} C_VEL
LIN {X 0,Y 262.354,Z 313.432,A -85,B 0,C 180,E1 -18613.349,E2 -18613.349} C_VEL
LIN {X 0,Y 263.953,Z 302.549,A -85,B 0,C 180,E1 -18614.955,E2 -18614.955} C_VEL
LIN {X 0,Y 264.506,Z 297.621,A -85,B 0,C 180,E1 -18615.578,E2 -18615.578} C_VEL
LIN {X 0,Y 262.459,Z 286.221,A -85,B 0,C 180,E1 -18617.044,E2 -18617.044} C_VEL
LIN {X 0,Y 259.447,Z 273.452,A -85,B 0,C 180,E1 -18618.404,E2 -18618.404} C_VEL
LIN {X 0,Y 255.546,Z 260.282,A -85,B 0,C 180,E1 -18619.554,E2 -18619.554} C_VEL
LIN {X 0,Y 255.29,Z 258.895,A -85,B 0,C 180,E1 -18619.694,E2 -18619.694} C_VEL
LIN {X 0,Y 255.549,Z 257.08,A -85,B 0,C 180,E1 -18622.098,E2 -18622.098} C_VEL
LIN {X 0,Y 255.761,Z 256.628,A -85,B 0,C 180,E1 -18623.691,E2 -18623.691} C_VEL
LIN {X 0,Y 256.461,Z 256.537,A -85,B 0,C 180,E1 -18628.431,E2 -18628.431} C_VEL
LIN {X 0,Y 256.717,Z 256.506,A -85,B 0,C 180,E1 -18630.002,E2 -18630.002} C_VEL
LIN {X 0,Y 256.488,Z 256.538,A -85,B 0,C 180,E1 -18633.143,E2 -18633.143} C_VEL
LIN {X 0,Y 256.527,Z 256.528,A -85,B 0,C 180,E1 -18637.875,E2 -18637.875} C_VEL
LIN {X 0,Y 256.299,Z 256.56,A -85,B 0,C 180,E1 -18641.068,E2 -18641.068} C_VEL
LIN {X 0,Y 256.289,Z 256.559,A -85,B 0,C 180,E1 -18645.917,E2 -18645.917} C_VEL
LIN {X 0,Y 256.222,Z 256.568,A -85,B 0,C 180,E1 -18650.892,E2 -18650.892} C_VEL
LIN {X 0,Y 256.18,Z 256.577,A -85,B 0,C 180,E1 -18655.141,E2 -18655.141} C_VEL
LIN {X 0,Y 256.106,Z 256.583,A -85,B 0,C 180,E1 -18659.602,E2 -18659.602} C_VEL
LIN {X 0,Y 256.078,Z 256.585,A -85,B 0,C 180,E1 -18663.293,E2 -18663.293} C_VEL
LIN {X 0,Y 256.133,Z 256.579,A -85,B 0,C 180,E1 -18667.281,E2 -18667.281} C_VEL
LIN {X 0,Y 256.098,Z 256.583,A -85,B 0,C 180,E1 -18671.197,E2 -18671.197} C_VEL
LIN {X 0,Y 256.072,Z 256.583,A -85,B 0,C 180,E1 -18675.529,E2 -18675.529} C_VEL
LIN {X 0,Y 256.082,Z 256.586,A -85,B 0,C 180,E1 -18678.806,E2 -18678.806} C_VEL
LIN {X 0,Y 256.153,Z 256.571,A -85,B 0,C 180,E1 -18682.875,E2 -18682.875} C_VEL
LIN {X 0,Y 256.084,Z 256.579,A -85,B 0,C 180,E1 -18686.713,E2 -18686.713} C_VEL
LIN {X 0,Y 256.135,Z 256.577,A -85,B 0,C 180,E1 -18691.41,E2 -18691.41} C_VEL
LIN {X 0,Y 256.169,Z 256.573,A -85,B 0,C 180,E1 -18695.702,E2 -18695.702} C_VEL
LIN {X 0,Y 256.169,Z 256.563,A -85,B 0,C 180,E1 -18699.108,E2 -18699.108} C_VEL
LIN {X 0,Y 256.304,Z 256.557,A -85,B 0,C 180,E1 -18704.088,E2 -18704.088} C_VEL
LIN {X 0,Y 256.3,Z 256.557,A -85,B 0,C 180,E1 -18707.331,E2 -18707.331} C_VEL
LIN {X 0,Y 256.51,Z 256.526,A -85,B 0,C 180,E1 -18712.129,E2 -18712.129} C_VEL
LIN {X 0,Y 256.503,Z 256.527,A -85,B 0,C 180,E1 -18716.861,E2 -18716.861} C_VEL
LIN {X 0,Y 256.765,Z 256.502,A -85,B 0,C 180,E1 -18720.002,E2 -18720.002} C_VEL
LIN {X 0,Y 256.5,Z 256.532,A -85,B 0,C 180,E1 -18723.144,E2 -18723.144} C_VEL
LIN {X 0,Y 256.507,Z 256.526,A -85,B 0,C 180,E1 -18727.876,E2 -18727.876} C_VEL
LIN {X 0,Y 256.294,Z 256.558,A -85,B 0,C 180,E1 -18732.675,E2 -18732.675} C_VEL
LIN {X 0,Y 256.293,Z 256.556,A -85,B 0,C 180,E1 -18736.304,E2 -18736.304} C_VEL
LIN {X 0,Y 256.168,Z 256.573,A -85,B 0,C 180,E1 -18741.121,E2 -18741.121} C_VEL
LIN {X 0,Y 256.199,Z 256.573,A -85,B 0,C 180,E1 -18745.14,E2 -18745.14} C_VEL
LIN {X 0,Y 256.114,Z 256.582,A -85,B 0,C 180,E1 -18749.602,E2 -18749.602} C_VEL
LIN {X 0,Y 256.1,Z 256.584,A -85,B 0,C 180,E1 -18751.493,E2 -18751.493} C_VEL
LIN {X 0,Y 255.402,Z 256.671,A -85,B 0,C 180,E1 -18752.805,E2 -18752.805} C_VEL
LIN {X 0,Y 252.543,Z 257.028,A -85,B 0,C 180,E1 -18754.945,E2 -18754.945} C_VEL
LIN {X 0,Y 250.141,Z 257.327,A -85,B 0,C 180,E1 -18756.687,E2 -18756.687} C_VEL
LIN {X 0,Y 249.122,Z 257.452,A -85,B 0,C 180,E1 -18758.038,E2 -18758.038} C_VEL
LIN {X 0,Y 249.043,Z 257.461,A -85,B 0,C 180,E1 -18758.495,E2 -18758.495} C_VEL
LIN {X 0,Y 249.099,Z 257.654,A -85,B 0,C 180,E1 -18759.912,E2 -18759.912} C_VEL
LIN {X 0,Y 249.638,Z 260.741,A -85,B 0,C 180,E1 -18762.946,E2 -18762.946} C_VEL
LIN {X 0,Y 250.56,Z 265.818,A -85,B 0,C 180,E1 -18767.685,E2 -18767.685} C_VEL
LIN {X 0,Y 251.305,Z 270.218,A -85,B 0,C 180,E1 -18771.544,E2 -18771.544} C_VEL
LIN {X 0,Y 251.183,Z 273.22,A -85,B 0,C 180,E1 -18774.013,E2 -18774.013} C_VEL
LIN {X 0,Y 250.148,Z 277.934,A -85,B 0,C 180,E1 -18777.735,E2 -18777.735} C_VEL
LIN {X 0,Y 248.943,Z 284.45,A -85,B 0,C 180,E1 -18782.726,E2 -18782.726} C_VEL
LIN {X 0,Y 251.433,Z 298.851,A -85,B 0,C 180,E1 -18783.781,E2 -18783.781} C_VEL
LIN {X 0,Y 253.153,Z 311.84,A -85,B 0,C 180,E1 -18785.018,E2 -18785.018} C_VEL
LIN {X 0,Y 254.128,Z 323.325,A -85,B 0,C 180,E1 -18786.363,E2 -18786.363} C_VEL
LIN {X 0,Y 254.681,Z 334.242,A -85,B 0,C 180,E1 -18787.913,E2 -18787.913} C_VEL
LIN {X 0,Y 254.315,Z 339.408,A -85,B 0,C 180,E1 -18788.732,E2 -18788.732} C_VEL
LIN {X 0,Y 252.551,Z 349.197,A -85,B 0,C 180,E1 -18790.49,E2 -18790.49} C_VEL
LIN {X 0,Y 250.864,Z 358.756,A -85,B 0,C 180,E1 -18792.629,E2 -18792.629} C_VEL
LIN {X 0,Y 249.489,Z 366.897,A -85,B 0,C 180,E1 -18794.895,E2 -18794.895} C_VEL
LIN {X 0,Y 248.296,Z 373.858,A -85,B 0,C 180,E1 -18797.327,E2 -18797.327} C_VEL
LIN {X 0,Y 247.514,Z 380.249,A -85,B 0,C 180,E1 -18800.189,E2 -18800.189} C_VEL
LIN {X 0,Y 247.168,Z 384.413,A -85,B 0,C 180,E1 -18802.647,E2 -18802.647} C_VEL
LIN {X 0,Y 247.095,Z 387.487,A -85,B 0,C 180,E1 -18805.104,E2 -18805.104} C_VEL
LIN {X 0,Y 247.155,Z 388.996,A -85,B 0,C 180,E1 -18806.738,E2 -18806.738} C_VEL
LIN {X 0,Y 247.149,Z 390.03,A -85,B 0,C 180,E1 -18808.369,E2 -18808.369} C_VEL
LIN {X 0,Y 247.204,Z 390.655,A -85,B 0,C 180,E1 -18809.998,E2 -18809.998} C_VEL
LIN {X 0,Y 247.116,Z 390.872,A -85,B 0,C 180,E1 -18811.628,E2 -18811.628} C_VEL
LIN {X 0,Y 247.049,Z 390.693,A -85,B 0,C 180,E1 -18813.26,E2 -18813.26} C_VEL
LIN {X 0,Y 246.99,Z 389.929,A -85,B 0,C 180,E1 -18815.165,E2 -18815.165} C_VEL
LIN {X 0,Y 247.199,Z 387.651,A -85,B 0,C 180,E1 -18818.171,E2 -18818.171} C_VEL
LIN {X 0,Y 247.718,Z 384.735,A -85,B 0,C 180,E1 -18820.625,E2 -18820.625} C_VEL
LIN {X 0,Y 248.571,Z 380.826,A -85,B 0,C 180,E1 -18823.071,E2 -18823.071} C_VEL
LIN {X 0,Y 250.069,Z 375.834,A -85,B 0,C 180,E1 -18825.484,E2 -18825.484} C_VEL
LIN {X 0,Y 251.879,Z 369.611,A -85,B 0,C 180,E1 -18827.872,E2 -18827.872} C_VEL
LIN {X 0,Y 253.997,Z 361.952,A -85,B 0,C 180,E1 -18830.233,E2 -18830.233} C_VEL
LIN {X 0,Y 256.727,Z 352.428,A -85,B 0,C 180,E1 -18832.534,E2 -18832.534} C_VEL
LIN {X 0,Y 259.359,Z 342.697,A -85,B 0,C 180,E1 -18834.407,E2 -18834.407} C_VEL
LIN {X 0,Y 260.002,Z 333.634,A -85,B 0,C 180,E1 -18836.026,E2 -18836.026} C_VEL
LIN {X 0,Y 259.944,Z 323.506,A -85,B 0,C 180,E1 -18837.643,E2 -18837.643} C_VEL
LIN {X 0,Y 258.713,Z 311.426,A -85,B 0,C 180,E1 -18839.402,E2 -18839.402} C_VEL
LIN {X 0,Y 256.31,Z 299.511,A -85,B 0,C 180,E1 -18841.019,E2 -18841.019} C_VEL
LIN {X 0,Y 252.989,Z 288.037,A -85,B 0,C 180,E1 -18842.521,E2 -18842.521} C_VEL
LIN {X 0,Y 251.953,Z 284.851,A -85,B 0,C 180,E1 -18842.918,E2 -18842.918} C_VEL
LIN {X 0,Y 250.986,Z 281.189,A -85,B 0,C 180,E1 -18843.352,E2 -18843.352} C_VEL
LIN {X 0,Y 252.019,Z 277.145,A -85,B 0,C 180,E1 -18846.836,E2 -18846.836} C_VEL
LIN {X 0,Y 252.042,Z 275.185,A -85,B 0,C 180,E1 -18848.667,E2 -18848.667} C_VEL
LIN {X 0,Y 251.583,Z 271.811,A -85,B 0,C 180,E1 -18852.099,E2 -18852.099} C_VEL
LIN {X 0,Y 250.819,Z 267.747,A -85,B 0,C 180,E1 -18856.76,E2 -18856.76} C_VEL
LIN {X 0,Y 250.413,Z 265.378,A -85,B 0,C 180,E1 -18859.794,E2 -18859.794} C_VEL
LIN {X 0,Y 249.941,Z 262.611,A -85,B 0,C 180,E1 -18863.806,E2 -18863.806} C_VEL
LIN {X 0,Y 249.54,Z 260.332,A -85,B 0,C 180,E1 -18867.659,E2 -18867.659} C_VEL
LIN {X 0,Y 249.289,Z 258.492,A -85,B 0,C 180,E1 -18871.36,E2 -18871.36} C_VEL
LIN {X 0,Y 249.129,Z 257.453,A -85,B 0,C 180,E1 -18874.515,E2 -18874.515} C_VEL
LIN {X 0,Y 249.093,Z 257.457,A -85,B 0,C 180,E1 -18878.598,E2 -18878.598} C_VEL
LIN {X 0,Y 249.238,Z 257.44,A -85,B 0,C 180,E1 -18883.619,E2 -18883.619} C_VEL
LIN {X 0,Y 249.249,Z 257.437,A -85,B 0,C 180,E1 -18888.614,E2 -18888.614} C_VEL
LIN {X 0,Y 249.479,Z 257.409,A -85,B 0,C 180,E1 -18891.9,E2 -18891.9} C_VEL
LIN {X 0,Y 249.433,Z 257.416,A -85,B 0,C 180,E1 -18896.767,E2 -18896.767} C_VEL
LIN {X 0,Y 249.729,Z 257.378,A -85,B 0,C 180,E1 -18899.997,E2 -18899.997} C_VEL
LIN {X 0,Y 249.431,Z 257.416,A -85,B 0,C 180,E1 -18903.228,E2 -18903.228} C_VEL
LIN {X 0,Y 249.456,Z 257.479,A -85,B 0,C 180,E1 -18906.776,E2 -18906.776} C_VEL
LIN {X 0,Y 249.559,Z 258.348,A -85,B 0,C 180,E1 -18909.725,E2 -18909.725} C_VEL
LIN {X 0,Y 249.58,Z 260.398,A -85,B 0,C 180,E1 -18914.678,E2 -18914.678} C_VEL
LIN {X 0,Y 249.535,Z 261.947,A -85,B 0,C 180,E1 -18918.045,E2 -18918.045} C_VEL
LIN {X 0,Y 249.529,Z 262.901,A -85,B 0,C 180,E1 -18919.537,E2 -18919.537} C_VEL
LIN {X 0,Y 250.7,Z 265.859,A -85,B 0,C 180,E1 -18919.975,E2 -18919.975} C_VEL
LIN {X 0,Y 251.889,Z 267.954,A -85,B 0,C 180,E1 -18920.356,E2 -18920.356} C_VEL
LIN {X 0,Y 256.232,Z 277.249,A -85,B 0,C 180,E1 -18921.948,E2 -18921.948} C_VEL
LIN {X 0,Y 260.006,Z 287.683,A -85,B 0,C 180,E1 -18923.718,E2 -18923.718} C_VEL
LIN {X 0,Y 262.828,Z 298.668,A -85,B 0,C 180,E1 -18925.61,E2 -18925.61} C_VEL
LIN {X 0,Y 264.124,Z 308.346,A -85,B 0,C 180,E1 -18927.357,E2 -18927.357} C_VEL
LIN {X 0,Y 261.852,Z 317.956,A -85,B 0,C 180,E1 -18928.886,E2 -18928.886} C_VEL
LIN {X 0,Y 259.477,Z 327.033,A -85,B 0,C 180,E1 -18930.675,E2 -18930.675} C_VEL
LIN {X 0,Y 256.98,Z 335.783,A -85,B 0,C 180,E1 -18932.812,E2 -18932.812} C_VEL
LIN {X 0,Y 254.679,Z 342.962,A -85,B 0,C 180,E1 -18934.987,E2 -18934.987} C_VEL
LIN {X 0,Y 252.765,Z 348.753,A -85,B 0,C 180,E1 -18937.186,E2 -18937.186} C_VEL
LIN {X 0,Y 251.154,Z 353.446,A -85,B 0,C 180,E1 -18939.424,E2 -18939.424} C_VEL
LIN {X 0,Y 249.87,Z 357.173,A -85,B 0,C 180,E1 -18941.707,E2 -18941.707} C_VEL
LIN {X 0,Y 248.383,Z 360.928,A -85,B 0,C 180,E1 -18944.981,E2 -18944.981} C_VEL
LIN {X 0,Y 247.634,Z 362.665,A -85,B 0,C 180,E1 -18947.548,E2 -18947.548} C_VEL
LIN {X 0,Y 247.163,Z 363.415,A -85,B 0,C 180,E1 -18950.146,E2 -18950.146} C_VEL
LIN {X 0,Y 246.936,Z 362.979,A -85,B 0,C 180,E1 -18953.298,E2 -18953.298} C_VEL
LIN {X 0,Y 247.007,Z 361.725,A -85,B 0,C 180,E1 -18955.596,E2 -18955.596} C_VEL
LIN {X 0,Y 247.43,Z 359.051,A -85,B 0,C 180,E1 -18958.437,E2 -18958.437} C_VEL
LIN {X 0,Y 248.143,Z 354.862,A -85,B 0,C 180,E1 -18961.395,E2 -18961.395} C_VEL
LIN {X 0,Y 248.929,Z 350.074,A -85,B 0,C 180,E1 -18963.873,E2 -18963.873} C_VEL
LIN {X 0,Y 250.085,Z 343.825,A -85,B 0,C 180,E1 -18966.395,E2 -18966.395} C_VEL
LIN {X 0,Y 251.38,Z 336.719,A -85,B 0,C 180,E1 -18968.69,E2 -18968.69} C_VEL
LIN {X 0,Y 252.944,Z 328.47,A -85,B 0,C 180,E1 -18970.844,E2 -18970.844} C_VEL
LIN {X 0,Y 254.597,Z 319.536,A -85,B 0,C 180,E1 -18972.74,E2 -18972.74} C_VEL
LIN {X 0,Y 256.287,Z 309.292,A -85,B 0,C 180,E1 -18974.494,E2 -18974.494} C_VEL
LIN {X 0,Y 257.639,Z 298.695,A -85,B 0,C 180,E1 -18975.967,E2 -18975.967} C_VEL
LIN {X 0,Y 255.7,Z 287.625,A -85,B 0,C 180,E1 -18977.453,E2 -18977.453} C_VEL
LIN {X 0,Y 253.01,Z 275.876,A -85,B 0,C 180,E1 -18978.789,E2 -18978.789} C_VEL
LIN {X 0,Y 249.371,Z 263.266,A -85,B 0,C 180,E1 -18979.972,E2 -18979.972} C_VEL
LIN {X 0,Y 248.272,Z 259.278,A -85,B 0,C 180,E1 -18980.326,E2 -18980.326} C_VEL
LIN {X 0,Y 248.462,Z 258.134,A -85,B 0,C 180,E1 -18981.871,E2 -18981.871} C_VEL
LIN {X 0,Y 248.68,Z 257.509,A -85,B 0,C 180,E1 -18983.511,E2 -18983.511} C_VEL
LIN {X 0,Y 249.401,Z 257.416,A -85,B 0,C 180,E1 -18988.387,E2 -18988.387} C_VEL
LIN {X 0,Y 249.676,Z 257.383,A -85,B 0,C 180,E1 -18990.002,E2 -18990.002} C_VEL
LIN {X 0,Y 249.664,Z 257.387,A -85,B 0,C 180,E1 -18991.615,E2 -18991.615} C_VEL
LIN {X 0,Y 249.449,Z 257.411,A -85,B 0,C 180,E1 -18996.472,E2 -18996.472} C_VEL
LIN {X 0,Y 249.377,Z 257.42,A -85,B 0,C 180,E1 -18999.737,E2 -18999.737} C_VEL
LIN {X 0,Y 249.195,Z 257.441,A -85,B 0,C 180,E1 -19004.706,E2 -19004.706} C_VEL
LIN {X 0,Y 249.139,Z 257.452,A -85,B 0,C 180,E1 -19008.079,E2 -19008.079} C_VEL
LIN {X 0,Y 249.126,Z 257.447,A -85,B 0,C 180,E1 -19011.516,E2 -19011.516} C_VEL
LIN {X 0,Y 249.122,Z 257.455,A -85,B 0,C 180,E1 -19015.485,E2 -19015.485} C_VEL
LIN {X 0,Y 249.076,Z 257.462,A -85,B 0,C 180,E1 -19018.996,E2 -19018.996} C_VEL
LIN {X 0,Y 249.029,Z 257.467,A -85,B 0,C 180,E1 -19022.428,E2 -19022.428} C_VEL
LIN {X 0,Y 249.068,Z 257.461,A -85,B 0,C 180,E1 -19026.341,E2 -19026.341} C_VEL
LIN {X 0,Y 249.072,Z 257.459,A -85,B 0,C 180,E1 -19030.467,E2 -19030.467} C_VEL
LIN {X 0,Y 249.018,Z 257.464,A -85,B 0,C 180,E1 -19034.878,E2 -19034.878} C_VEL
LIN {X 0,Y 249.048,Z 257.46,A -85,B 0,C 180,E1 -19037.374,E2 -19037.374} C_VEL
LIN {X 0,Y 249.049,Z 257.458,A -85,B 0,C 180,E1 -19041.627,E2 -19041.627} C_VEL
LIN {X 0,Y 249.06,Z 257.447,A -85,B 0,C 180,E1 -19045.646,E2 -19045.646} C_VEL
LIN {X 0,Y 249.05,Z 257.457,A -85,B 0,C 180,E1 -19049.476,E2 -19049.476} C_VEL
LIN {X 0,Y 249.073,Z 257.457,A -85,B 0,C 180,E1 -19053.165,E2 -19053.165} C_VEL
LIN {X 0,Y 249.081,Z 257.451,A -85,B 0,C 180,E1 -19056.736,E2 -19056.736} C_VEL
LIN {X 0,Y 249.113,Z 257.443,A -85,B 0,C 180,E1 -19060.215,E2 -19060.215} C_VEL
LIN {X 0,Y 249.246,Z 257.433,A -85,B 0,C 180,E1 -19063.625,E2 -19063.625} C_VEL
LIN {X 0,Y 249.25,Z 257.435,A -85,B 0,C 180,E1 -19068.619,E2 -19068.619} C_VEL
LIN {X 0,Y 249.452,Z 257.406,A -85,B 0,C 180,E1 -19071.905,E2 -19071.905} C_VEL
LIN {X 0,Y 249.298,Z 257.419,A -85,B 0,C 180,E1 -19075.151,E2 -19075.151} C_VEL
LIN {X 0,Y 249.682,Z 257.381,A -85,B 0,C 180,E1 -19078.39,E2 -19078.39} C_VEL
LIN {X 0,Y 249.681,Z 257.385,A -85,B 0,C 180,E1 -19081.615,E2 -19081.615} C_VEL
LIN {X 0,Y 249.448,Z 257.403,A -85,B 0,C 180,E1 -19086.473,E2 -19086.473} C_VEL
LIN {X 0,Y 249.351,Z 257.421,A -85,B 0,C 180,E1 -19089.739,E2 -19089.739} C_VEL
LIN {X 0,Y 249.215,Z 257.44,A -85,B 0,C 180,E1 -19094.705,E2 -19094.705} C_VEL
LIN {X 0,Y 249.149,Z 257.442,A -85,B 0,C 180,E1 -19098.079,E2 -19098.079} C_VEL
LIN {X 0,Y 249.098,Z 257.457,A -85,B 0,C 180,E1 -19101.52,E2 -19101.52} C_VEL
LIN {X 0,Y 249.141,Z 257.45,A -85,B 0,C 180,E1 -19105.483,E2 -19105.483} C_VEL
LIN {X 0,Y 249.084,Z 257.455,A -85,B 0,C 180,E1 -19108.99,E2 -19108.99} C_VEL
LIN {X 0,Y 249.041,Z 257.462,A -85,B 0,C 180,E1 -19112.427,E2 -19112.427} C_VEL
LIN {X 0,Y 249.04,Z 257.461,A -85,B 0,C 180,E1 -19116.346,E2 -19116.346} C_VEL
LIN {X 0,Y 249.043,Z 257.461,A -85,B 0,C 180,E1 -19118.495,E2 -19118.495} C_VEL
LIN {X 0,Y 248.445,Z 258.001,A -85,B 0,C 180,E1 -19119.84,E2 -19119.84} C_VEL
LIN {X 0,Y 247.034,Z 259.288,A -85,B 0,C 180,E1 -19121.144,E2 -19121.144} C_VEL
LIN {X 0,Y 243.835,Z 262.506,A -85,B 0,C 180,E1 -19123.74,E2 -19123.74} C_VEL
LIN {X 0,Y 243.082,Z 264.059,A -85,B 0,C 180,E1 -19125.085,E2 -19125.085} C_VEL
LIN {X 0,Y 243.094,Z 264.544,A -85,B 0,C 180,E1 -19125.54,E2 -19125.54} C_VEL
LIN {X 0,Y 243.922,Z 268.958,A -85,B 0,C 180,E1 -19129.643,E2 -19129.643} C_VEL
LIN {X 0,Y 244.323,Z 272.599,A -85,B 0,C 180,E1 -19132.836,E2 -19132.836} C_VEL
LIN {X 0,Y 243.658,Z 276.166,A -85,B 0,C 180,E1 -19135.773,E2 -19135.773} C_VEL
LIN {X 0,Y 242.349,Z 282.025,A -85,B 0,C 180,E1 -19140.461,E2 -19140.461} C_VEL
LIN {X 0,Y 241.998,Z 284.065,A -85,B 0,C 180,E1 -19142.075,E2 -19142.075} C_VEL
LIN {X 0,Y 244.435,Z 298.009,A -85,B 0,C 180,E1 -19143.117,E2 -19143.117} C_VEL
LIN {X 0,Y 246.234,Z 311.609,A -85,B 0,C 180,E1 -19144.456,E2 -19144.456} C_VEL
LIN {X 0,Y 247.248,Z 323.843,A -85,B 0,C 180,E1 -19145.947,E2 -19145.947} C_VEL
LIN {X 0,Y 247.741,Z 335.498,A -85,B 0,C 180,E1 -19147.7,E2 -19147.7} C_VEL
LIN {X 0,Y 247.278,Z 340.498,A -85,B 0,C 180,E1 -19148.534,E2 -19148.534} C_VEL
LIN {X 0,Y 245.476,Z 350.038,A -85,B 0,C 180,E1 -19150.34,E2 -19150.34} C_VEL
LIN {X 0,Y 243.79,Z 359.331,A -85,B 0,C 180,E1 -19152.526,E2 -19152.526} C_VEL
LIN {X 0,Y 242.38,Z 367.292,A -85,B 0,C 180,E1 -19154.871,E2 -19154.871} C_VEL
LIN {X 0,Y 241.159,Z 374.103,A -85,B 0,C 180,E1 -19157.373,E2 -19157.373} C_VEL
LIN {X 0,Y 240.471,Z 379.552,A -85,B 0,C 180,E1 -19159.899,E2 -19159.899} C_VEL
LIN {X 0,Y 240.116,Z 383.787,A -85,B 0,C 180,E1 -19162.43,E2 -19162.43} C_VEL
LIN {X 0,Y 240.02,Z 386.924,A -85,B 0,C 180,E1 -19164.959,E2 -19164.959} C_VEL
LIN {X 0,Y 240.063,Z 388.467,A -85,B 0,C 180,E1 -19166.642,E2 -19166.642} C_VEL
LIN {X 0,Y 240.075,Z 389.557,A -85,B 0,C 180,E1 -19168.321,E2 -19168.321} C_VEL
LIN {X 0,Y 240.125,Z 390.21,A -85,B 0,C 180,E1 -19169.998,E2 -19169.998} C_VEL
LIN {X 0,Y 240.041,Z 390.454,A -85,B 0,C 180,E1 -19171.676,E2 -19171.676} C_VEL
LIN {X 0,Y 239.962,Z 390.304,A -85,B 0,C 180,E1 -19173.356,E2 -19173.356} C_VEL
LIN {X 0,Y 239.919,Z 389.696,A -85,B 0,C 180,E1 -19175.125,E2 -19175.125} C_VEL
LIN {X 0,Y 240.154,Z 387.379,A -85,B 0,C 180,E1 -19178.412,E2 -19178.412} C_VEL
LIN {X 0,Y 240.699,Z 384.537,A -85,B 0,C 180,E1 -19180.939,E2 -19180.939} C_VEL
LIN {X 0,Y 241.632,Z 380.701,A -85,B 0,C 180,E1 -19183.453,E2 -19183.453} C_VEL
LIN {X 0,Y 243.216,Z 375.783,A -85,B 0,C 180,E1 -19185.931,E2 -19185.931} C_VEL
LIN {X 0,Y 245.13,Z 369.64,A -85,B 0,C 180,E1 -19188.382,E2 -19188.382} C_VEL
LIN {X 0,Y 247.333,Z 362.077,A -85,B 0,C 180,E1 -19190.803,E2 -19190.803} C_VEL
LIN {X 0,Y 249.672,Z 354.458,A -85,B 0,C 180,E1 -19192.769,E2 -19192.769} C_VEL
LIN {X 0,Y 252.694,Z 344.265,A -85,B 0,C 180,E1 -19194.875,E2 -19194.875} C_VEL
LIN {X 0,Y 253.577,Z 334.542,A -85,B 0,C 180,E1 -19196.706,E2 -19196.706} C_VEL
LIN {X 0,Y 253.632,Z 324.48,A -85,B 0,C 180,E1 -19198.395,E2 -19198.395} C_VEL
LIN {X 0,Y 252.689,Z 313.88,A -85,B 0,C 180,E1 -19200.04,E2 -19200.04} C_VEL
LIN {X 0,Y 250.919,Z 303.693,A -85,B 0,C 180,E1 -19201.537,E2 -19201.537} C_VEL
LIN {X 0,Y 247.811,Z 291.85,A -85,B 0,C 180,E1 -19203.209,E2 -19203.209} C_VEL
LIN {X 0,Y 245.505,Z 284.648,A -85,B 0,C 180,E1 -19204.206,E2 -19204.206} C_VEL
LIN {X 0,Y 244.436,Z 281.642,A -85,B 0,C 180,E1 -19204.622,E2 -19204.622} C_VEL
LIN {X 0,Y 244.352,Z 280.644,A -85,B 0,C 180,E1 -19204.764,E2 -19204.764} C_VEL
LIN {X 0,Y 245.021,Z 278.112,A -85,B 0,C 180,E1 -19207.036,E2 -19207.036} C_VEL
LIN {X 0,Y 244.967,Z 275.863,A -85,B 0,C 180,E1 -19209.226,E2 -19209.226} C_VEL
LIN {X 0,Y 244.673,Z 273.533,A -85,B 0,C 180,E1 -19211.681,E2 -19211.681} C_VEL
LIN {X 0,Y 243.937,Z 269.603,A -85,B 0,C 180,E1 -19216.252,E2 -19216.252} C_VEL
LIN {X 0,Y 243.373,Z 266.353,A -85,B 0,C 180,E1 -19220.555,E2 -19220.555} C_VEL
LIN {X 0,Y 242.949,Z 263.665,A -85,B 0,C 180,E1 -19224.648,E2 -19224.648} C_VEL
LIN {X 0,Y 242.526,Z 261.516,A -85,B 0,C 180,E1 -19228.557,E2 -19228.557} C_VEL
LIN {X 0,Y 242.277,Z 259.768,A -85,B 0,C 180,E1 -19232.344,E2 -19232.344} C_VEL
LIN {X 0,Y 242.055,Z 258.419,A -85,B 0,C 180,E1 -19236.013,E2 -19236.013} C_VEL
LIN {X 0,Y 242.035,Z 258.337,A -85,B 0,C 180,E1 -19239.605,E2 -19239.605} C_VEL
LIN {X 0,Y 242.16,Z 258.32,A -85,B 0,C 180,E1 -19243.275,E2 -19243.275} C_VEL
LIN {X 0,Y 242.183,Z 258.318,A -85,B 0,C 180,E1 -19248.277,E2 -19248.277} C_VEL
LIN {X 0,Y 242.43,Z 258.287,A -85,B 0,C 180,E1 -19251.663,E2 -19251.663} C_VEL
LIN {X 0,Y 242.257,Z 258.31,A -85,B 0,C 180,E1 -19255.005,E2 -19255.005} C_VEL
LIN {X 0,Y 242.631,Z 258.262,A -85,B 0,C 180,E1 -19258.338,E2 -19258.338} C_VEL
LIN {X 0,Y 242.631,Z 258.264,A -85,B 0,C 180,E1 -19261.657,E2 -19261.657} C_VEL
LIN {X 0,Y 242.258,Z 258.329,A -85,B 0,C 180,E1 -19264.99,E2 -19264.99} C_VEL
LIN {X 0,Y 242.582,Z 259.302,A -85,B 0,C 180,E1 -19268.326,E2 -19268.326} C_VEL
LIN {X 0,Y 242.543,Z 260.542,A -85,B 0,C 180,E1 -19271.7,E2 -19271.7} C_VEL
LIN {X 0,Y 242.617,Z 261.936,A -85,B 0,C 180,E1 -19275.109,E2 -19275.109} C_VEL
LIN {X 0,Y 242.555,Z 263.256,A -85,B 0,C 180,E1 -19278.036,E2 -19278.036} C_VEL
LIN {X 0,Y 243.733,Z 266.356,A -85,B 0,C 180,E1 -19278.521,E2 -19278.521} C_VEL
LIN {X 0,Y 245.048,Z 268.298,A -85,B 0,C 180,E1 -19278.948,E2 -19278.948} C_VEL
LIN {X 0,Y 250.165,Z 279.238,A -85,B 0,C 180,E1 -19280.986,E2 -19280.986} C_VEL
LIN {X 0,Y 254.102,Z 290.263,A -85,B 0,C 180,E1 -19282.993,E2 -19282.993} C_VEL
LIN {X 0,Y 256.595,Z 300.57,A -85,B 0,C 180,E1 -19284.902,E2 -19284.902} C_VEL
LIN {X 0,Y 257.815,Z 308.965,A -85,B 0,C 180,E1 -19286.509,E2 -19286.509} C_VEL
LIN {X 0,Y 257.496,Z 311.447,A -85,B 0,C 180,E1 -19286.927,E2 -19286.927} C_VEL
LIN {X 0,Y 255.107,Z 320.841,A -85,B 0,C 180,E1 -19288.535,E2 -19288.535} C_VEL
LIN {X 0,Y 252.622,Z 329.708,A -85,B 0,C 180,E1 -19290.413,E2 -19290.413} C_VEL
LIN {X 0,Y 250.095,Z 337.788,A -85,B 0,C 180,E1 -19292.541,E2 -19292.541} C_VEL
LIN {X 0,Y 247.293,Z 345.809,A -85,B 0,C 180,E1 -19295.211,E2 -19295.211} C_VEL
LIN {X 0,Y 245.061,Z 352.144,A -85,B 0,C 180,E1 -19297.963,E2 -19297.963} C_VEL
LIN {X 0,Y 243.543,Z 356.219,A -85,B 0,C 180,E1 -19300.265,E2 -19300.265} C_VEL
LIN {X 0,Y 242.755,Z 358.317,A -85,B 0,C 180,E1 -19301.745,E2 -19301.745} C_VEL
LIN {X 0,Y 241.551,Z 361.108,A -85,B 0,C 180,E1 -19304.285,E2 -19304.285} C_VEL
LIN {X 0,Y 240.72,Z 362.93,A -85,B 0,C 180,E1 -19306.873,E2 -19306.873} C_VEL
LIN {X 0,Y 240.107,Z 363.829,A -85,B 0,C 180,E1 -19309.916,E2 -19309.916} C_VEL
LIN {X 0,Y 239.869,Z 363.67,A -85,B 0,C 180,E1 -19312.282,E2 -19312.282} C_VEL
LIN {X 0,Y 239.888,Z 362.42,A -85,B 0,C 180,E1 -19315.111,E2 -19315.111} C_VEL
LIN {X 0,Y 240.284,Z 359.689,A -85,B 0,C 180,E1 -19318.234,E2 -19318.234} C_VEL
LIN {X 0,Y 240.942,Z 355.955,A -85,B 0,C 180,E1 -19321.046,E2 -19321.046} C_VEL
LIN {X 0,Y 241.946,Z 350.092,A -85,B 0,C 180,E1 -19324.214,E2 -19324.214} C_VEL
LIN {X 0,Y 243.202,Z 343.675,A -85,B 0,C 180,E1 -19326.833,E2 -19326.833} C_VEL
LIN {X 0,Y 244.739,Z 335.722,A -85,B 0,C 180,E1 -19329.406,E2 -19329.406} C_VEL
LIN {X 0,Y 246.461,Z 326.656,A -85,B 0,C 180,E1 -19331.721,E2 -19331.721} C_VEL
LIN {X 0,Y 248.425,Z 316.199,A -85,B 0,C 180,E1 -19333.85,E2 -19333.85} C_VEL
LIN {X 0,Y 250.125,Z 305.67,A -85,B 0,C 180,E1 -19335.562,E2 -19335.562} C_VEL
LIN {X 0,Y 250.824,Z 300.874,A -85,B 0,C 180,E1 -19336.223,E2 -19336.223} C_VEL
LIN {X 0,Y 249.533,Z 291.863,A -85,B 0,C 180,E1 -19337.513,E2 -19337.513} C_VEL
LIN {X 0,Y 247.047,Z 280.282,A -85,B 0,C 180,E1 -19338.948,E2 -19338.948} C_VEL
LIN {X 0,Y 243.516,Z 267.224,A -85,B 0,C 180,E1 -19340.29,E2 -19340.29} C_VEL
LIN {X 0,Y 241.295,Z 259.672,A -85,B 0,C 180,E1 -19340.97,E2 -19340.97} C_VEL
LIN {X 0,Y 241.582,Z 258.393,A -85,B 0,C 180,E1 -19343.319,E2 -19343.319} C_VEL
LIN {X 0,Y 242.343,Z 258.295,A -85,B 0,C 180,E1 -19348.34,E2 -19348.34} C_VEL
LIN {X 0,Y 242.634,Z 258.26,A -85,B 0,C 180,E1 -19350.002,E2 -19350.002} C_VEL
LIN {X 0,Y 242.624,Z 258.264,A -85,B 0,C 180,E1 -19351.662,E2 -19351.662} C_VEL
LIN {X 0,Y 242.421,Z 258.287,A -85,B 0,C 180,E1 -19356.661,E2 -19356.661} C_VEL
LIN {X 0,Y 242.302,Z 258.3,A -85,B 0,C 180,E1 -19360.024,E2 -19360.024} C_VEL
LIN {X 0,Y 242.156,Z 258.32,A -85,B 0,C 180,E1 -19365.143,E2 -19365.143} C_VEL
LIN {X 0,Y 242.08,Z 258.333,A -85,B 0,C 180,E1 -19368.625,E2 -19368.625} C_VEL
LIN {X 0,Y 242.054,Z 258.327,A -85,B 0,C 180,E1 -19372.178,E2 -19372.178} C_VEL
LIN {X 0,Y 242.058,Z 258.334,A -85,B 0,C 180,E1 -19375.841,E2 -19375.841} C_VEL
LIN {X 0,Y 242.022,Z 258.338,A -85,B 0,C 180,E1 -19379.583,E2 -19379.583} C_VEL
LIN {X 0,Y 241.984,Z 258.34,A -85,B 0,C 180,E1 -19383.494,E2 -19383.494} C_VEL
LIN {X 0,Y 242.006,Z 258.338,A -85,B 0,C 180,E1 -19387.581,E2 -19387.581} C_VEL
LIN {X 0,Y 241.98,Z 258.342,A -85,B 0,C 180,E1 -19391.915,E2 -19391.915} C_VEL
LIN {X 0,Y 241.982,Z 258.343,A -85,B 0,C 180,E1 -19396.562,E2 -19396.562} C_VEL
LIN {X 0,Y 241.986,Z 258.343,A -85,B 0,C 180,E1 -19400.291,E2 -19400.291} C_VEL
LIN {X 0,Y 242.035,Z 258.324,A -85,B 0,C 180,E1 -19404.501,E2 -19404.501} C_VEL
LIN {X 0,Y 241.976,Z 258.34,A -85,B 0,C 180,E1 -19408.483,E2 -19408.483} C_VEL
LIN {X 0,Y 242.008,Z 258.341,A -85,B 0,C 180,E1 -19412.316,E2 -19412.316} C_VEL
LIN {X 0,Y 242.059,Z 258.331,A -85,B 0,C 180,E1 -19416.019,E2 -19416.019} C_VEL
LIN {X 0,Y 242.04,Z 258.322,A -85,B 0,C 180,E1 -19419.611,E2 -19419.611} C_VEL
LIN {X 0,Y 242.167,Z 258.313,A -85,B 0,C 180,E1 -19423.281,E2 -19423.281} C_VEL
LIN {X 0,Y 242.186,Z 258.316,A -85,B 0,C 180,E1 -19428.283,E2 -19428.283} C_VEL
LIN {X 0,Y 242.399,Z 258.286,A -85,B 0,C 180,E1 -19431.667,E2 -19431.667} C_VEL
LIN {X 0,Y 242.258,Z 258.294,A -85,B 0,C 180,E1 -19435.01,E2 -19435.01} C_VEL
LIN {X 0,Y 242.642,Z 258.258,A -85,B 0,C 180,E1 -19438.343,E2 -19438.343} C_VEL
LIN {X 0,Y 242.642,Z 258.262,A -85,B 0,C 180,E1 -19441.662,E2 -19441.662} C_VEL
LIN {X 0,Y 242.419,Z 258.278,A -85,B 0,C 180,E1 -19446.662,E2 -19446.662} C_VEL
LIN {X 0,Y 242.276,Z 258.303,A -85,B 0,C 180,E1 -19450.026,E2 -19450.026} C_VEL
LIN {X 0,Y 242.176,Z 258.318,A -85,B 0,C 180,E1 -19455.143,E2 -19455.143} C_VEL
LIN {X 0,Y 242.083,Z 258.321,A -85,B 0,C 180,E1 -19458.626,E2 -19458.626} C_VEL
LIN {X 0,Y 242.024,Z 258.336,A -85,B 0,C 180,E1 -19462.181,E2 -19462.181} C_VEL
LIN {X 0,Y 242.077,Z 258.328,A -85,B 0,C 180,E1 -19465.839,E2 -19465.839} C_VEL
LIN {X 0,Y 242.018,Z 258.338,A -85,B 0,C 180,E1 -19469.584,E2 -19469.584} C_VEL
LIN {X 0,Y 241.991,Z 258.341,A -85,B 0,C 180,E1 -19473.493,E2 -19473.493} C_VEL
LIN {X 0,Y 241.999,Z 258.34,A -85,B 0,C 180,E1 -19477.583,E2 -19477.583} C_VEL
LIN {X 0,Y 242.08,Z 258.499,A -85,B 0,C 180,E1 -19479.509,E2 -19479.509} C_VEL
LIN {X 0,Y 242.817,Z 262.943,A -85,B 0,C 180,E1 -19484.002,E2 -19484.002} C_VEL
LIN {X 0,Y 243.094,Z 264.544,A -85,B 0,C 180,E1 -19485.54,E2 -19485.54} C_VEL
LIN {X 0,Y 242.71,Z 266.055,A -85,B 0,C 180,E1 -19486.882,E2 -19486.882} C_VEL
LIN {X 0,Y 240.291,Z 268.809,A -85,B 0,C 180,E1 -19489.068,E2 -19489.068} C_VEL
LIN {X 0,Y 237.421,Z 272.191,A -85,B 0,C 180,E1 -19491.753,E2 -19491.753} C_VEL
LIN {X 0,Y 237.168,Z 273.271,A -85,B 0,C 180,E1 -19492.68,E2 -19492.68} C_VEL
LIN {X 0,Y 236.605,Z 276.725,A -85,B 0,C 180,E1 -19495.64,E2 -19495.64} C_VEL
LIN {X 0,Y 235.124,Z 283.212,A -85,B 0,C 180,E1 -19500.976,E2 -19500.976} C_VEL
LIN {X 0,Y 235.038,Z 283.997,A -85,B 0,C 180,E1 -19501.416,E2 -19501.416} C_VEL
LIN {X 0,Y 237.459,Z 297.452,A -85,B 0,C 180,E1 -19502.46,E2 -19502.46} C_VEL
LIN {X 0,Y 239.134,Z 309.861,A -85,B 0,C 180,E1 -19503.702,E2 -19503.702} C_VEL
LIN {X 0,Y 240.19,Z 321.329,A -85,B 0,C 180,E1 -19505.108,E2 -19505.108} C_VEL
LIN {X 0,Y 240.766,Z 332.704,A -85,B 0,C 180,E1 -19506.79,E2 -19506.79} C_VEL
LIN {X 0,Y 240.601,Z 339.237,A -85,B 0,C 180,E1 -19507.907,E2 -19507.907} C_VEL
LIN {X 0,Y 238.744,Z 348.923,A -85,B 0,C 180,E1 -19509.762,E2 -19509.762} C_VEL
LIN {X 0,Y 237.024,Z 357.461,A -85,B 0,C 180,E1 -19511.774,E2 -19511.774} C_VEL
LIN {X 0,Y 235.96,Z 363.751,A -85,B 0,C 180,E1 -19513.562,E2 -19513.562} C_VEL
LIN {X 0,Y 234.611,Z 371.2,A -85,B 0,C 180,E1 -19516.133,E2 -19516.133} C_VEL
LIN {X 0,Y 233.634,Z 377.166,A -85,B 0,C 180,E1 -19518.723,E2 -19518.723} C_VEL
LIN {X 0,Y 233.161,Z 381.869,A -85,B 0,C 180,E1 -19521.33,E2 -19521.33} C_VEL
LIN {X 0,Y 233.037,Z 385.968,A -85,B 0,C 180,E1 -19524.417,E2 -19524.417} C_VEL
LIN {X 0,Y 232.975,Z 387.931,A -85,B 0,C 180,E1 -19526.539,E2 -19526.539} C_VEL
LIN {X 0,Y 233.003,Z 389.076,A -85,B 0,C 180,E1 -19528.27,E2 -19528.27} C_VEL
LIN {X 0,Y 233.048,Z 389.762,A -85,B 0,C 180,E1 -19529.998,E2 -19529.998} C_VEL
LIN {X 0,Y 232.966,Z 390.036,A -85,B 0,C 180,E1 -19531.727,E2 -19531.727} C_VEL
LIN {X 0,Y 232.812,Z 389.474,A -85,B 0,C 180,E1 -19534.985,E2 -19534.985} C_VEL
LIN {X 0,Y 232.907,Z 388.462,A -85,B 0,C 180,E1 -19536.931,E2 -19536.931} C_VEL
LIN {X 0,Y 233.464,Z 385.375,A -85,B 0,C 180,E1 -19540.404,E2 -19540.404} C_VEL
LIN {X 0,Y 234.3,Z 381.94,A -85,B 0,C 180,E1 -19542.999,E2 -19542.999} C_VEL
LIN {X 0,Y 235.777,Z 377.468,A -85,B 0,C 180,E1 -19545.56,E2 -19545.56} C_VEL
LIN {X 0,Y 238.007,Z 370.828,A -85,B 0,C 180,E1 -19548.506,E2 -19548.506} C_VEL
LIN {X 0,Y 240.295,Z 363.631,A -85,B 0,C 180,E1 -19550.993,E2 -19550.993} C_VEL
LIN {X 0,Y 243.166,Z 354.773,A -85,B 0,C 180,E1 -19553.414,E2 -19553.414} C_VEL
LIN {X 0,Y 246.25,Z 344.8,A -85,B 0,C 180,E1 -19555.572,E2 -19555.572} C_VEL
LIN {X 0,Y 247.207,Z 335.54,A -85,B 0,C 180,E1 -19557.402,E2 -19557.402} C_VEL
LIN {X 0,Y 247.372,Z 325.546,A -85,B 0,C 180,E1 -19559.186,E2 -19559.186} C_VEL
LIN {X 0,Y 246.376,Z 313.529,A -85,B 0,C 180,E1 -19561.152,E2 -19561.152} C_VEL
LIN {X 0,Y 244.486,Z 303.074,A -85,B 0,C 180,E1 -19562.776,E2 -19562.776} C_VEL
LIN {X 0,Y 241.397,Z 291.373,A -85,B 0,C 180,E1 -19564.562,E2 -19564.562} C_VEL
LIN {X 0,Y 238.997,Z 284.261,A -85,B 0,C 180,E1 -19565.642,E2 -19565.642} C_VEL
LIN {X 0,Y 237.831,Z 280.883,A -85,B 0,C 180,E1 -19566.133,E2 -19566.133} C_VEL
LIN {X 0,Y 237.748,Z 280.132,A -85,B 0,C 180,E1 -19566.241,E2 -19566.241} C_VEL
LIN {X 0,Y 238.08,Z 277.981,A -85,B 0,C 180,E1 -19568.307,E2 -19568.307} C_VEL
LIN {X 0,Y 237.554,Z 274.317,A -85,B 0,C 180,E1 -19572.298,E2 -19572.298} C_VEL
LIN {X 0,Y 236.86,Z 270.492,A -85,B 0,C 180,E1 -19576.962,E2 -19576.962} C_VEL
LIN {X 0,Y 236.362,Z 267.318,A -85,B 0,C 180,E1 -19581.358,E2 -19581.358} C_VEL
LIN {X 0,Y 235.908,Z 264.749,A -85,B 0,C 180,E1 -19585.523,E2 -19585.523} C_VEL
LIN {X 0,Y 235.525,Z 262.524,A -85,B 0,C 180,E1 -19589.919,E2 -19589.919} C_VEL
LIN {X 0,Y 235.29,Z 260.94,A -85,B 0,C 180,E1 -19593.644,E2 -19593.644} C_VEL
LIN {X 0,Y 235.05,Z 259.552,A -85,B 0,C 180,E1 -19597.951,E2 -19597.951} C_VEL
LIN {X 0,Y 235.006,Z 259.213,A -85,B 0,C 180,E1 -19600.792,E2 -19600.792} C_VEL
LIN {X 0,Y 235.111,Z 259.198,A -85,B 0,C 180,E1 -19604.391,E2 -19604.391} C_VEL
LIN {X 0,Y 235.337,Z 259.17,A -85,B 0,C 180,E1 -19610.219,E2 -19610.219} C_VEL
LIN {X 0,Y 235.401,Z 259.162,A -85,B 0,C 180,E1 -19613.139,E2 -19613.139} C_VEL
LIN {X 0,Y 235.591,Z 259.139,A -85,B 0,C 180,E1 -19618.288,E2 -19618.288} C_VEL
LIN {X 0,Y 235.591,Z 259.141,A -85,B 0,C 180,E1 -19621.707,E2 -19621.707} C_VEL
LIN {X 0,Y 235.562,Z 260.322,A -85,B 0,C 180,E1 -19626.851,E2 -19626.851} C_VEL
LIN {X 0,Y 235.623,Z 261.436,A -85,B 0,C 180,E1 -19630.307,E2 -19630.307} C_VEL
LIN {X 0,Y 235.641,Z 263.48,A -85,B 0,C 180,E1 -19635.568,E2 -19635.568} C_VEL
LIN {X 0,Y 235.65,Z 263.846,A -85,B 0,C 180,E1 -19636.4,E2 -19636.4} C_VEL
LIN {X 0,Y 236.92,Z 267.039,A -85,B 0,C 180,E1 -19636.973,E2 -19636.973} C_VEL
LIN {X 0,Y 238.357,Z 269.165,A -85,B 0,C 180,E1 -19637.489,E2 -19637.489} C_VEL
LIN {X 0,Y 242.488,Z 277.487,A -85,B 0,C 180,E1 -19639.204,E2 -19639.204} C_VEL
LIN {X 0,Y 246.081,Z 286.337,A -85,B 0,C 180,E1 -19640.968,E2 -19640.968} C_VEL
LIN {X 0,Y 249.003,Z 295.881,A -85,B 0,C 180,E1 -19642.832,E2 -19642.832} C_VEL
LIN {X 0,Y 251.007,Z 305.876,A -85,B 0,C 180,E1 -19644.831,E2 -19644.831} C_VEL
LIN {X 0,Y 251.589,Z 311.274,A -85,B 0,C 180,E1 -19645.948,E2 -19645.948} C_VEL
LIN {X 0,Y 249.022,Z 321.259,A -85,B 0,C 180,E1 -19647.693,E2 -19647.693} C_VEL
LIN {X 0,Y 246.091,Z 331.062,A -85,B 0,C 180,E1 -19649.838,E2 -19649.838} C_VEL
LIN {X 0,Y 243.168,Z 339.856,A -85,B 0,C 180,E1 -19652.291,E2 -19652.291} C_VEL
LIN {X 0,Y 240.317,Z 347.538,A -85,B 0,C 180,E1 -19655.033,E2 -19655.033} C_VEL
LIN {X 0,Y 237.972,Z 353.599,A -85,B 0,C 180,E1 -19657.901,E2 -19657.901} C_VEL
LIN {X 0,Y 236.096,Z 358.313,A -85,B 0,C 180,E1 -19660.907,E2 -19660.907} C_VEL
LIN {X 0,Y 234.557,Z 361.661,A -85,B 0,C 180,E1 -19664.022,E2 -19664.022} C_VEL
LIN {X 0,Y 233.792,Z 363.206,A -85,B 0,C 180,E1 -19666.261,E2 -19666.261} C_VEL
LIN {X 0,Y 233.182,Z 364.141,A -85,B 0,C 180,E1 -19668.889,E2 -19668.889} C_VEL
LIN {X 0,Y 232.822,Z 364.144,A -85,B 0,C 180,E1 -19671.7,E2 -19671.7} C_VEL
LIN {X 0,Y 232.809,Z 362.824,A -85,B 0,C 180,E1 -19675.003,E2 -19675.003} C_VEL
LIN {X 0,Y 233.075,Z 360.763,A -85,B 0,C 180,E1 -19677.59,E2 -19677.59} C_VEL
LIN {X 0,Y 233.747,Z 357.005,A -85,B 0,C 180,E1 -19680.677,E2 -19680.677} C_VEL
LIN {X 0,Y 234.487,Z 352.668,A -85,B 0,C 180,E1 -19683.285,E2 -19683.285} C_VEL
LIN {X 0,Y 235.75,Z 346.177,A -85,B 0,C 180,E1 -19686.271,E2 -19686.271} C_VEL
LIN {X 0,Y 237.12,Z 339.404,A -85,B 0,C 180,E1 -19688.713,E2 -19688.713} C_VEL
LIN {X 0,Y 238.756,Z 331.098,A -85,B 0,C 180,E1 -19691.109,E2 -19691.109} C_VEL
LIN {X 0,Y 240.666,Z 321.71,A -85,B 0,C 180,E1 -19693.284,E2 -19693.284} C_VEL
LIN {X 0,Y 242.596,Z 310.759,A -85,B 0,C 180,E1 -19695.318,E2 -19695.318} C_VEL
LIN {X 0,Y 244.016,Z 301.662,A -85,B 0,C 180,E1 -19696.68,E2 -19696.68} C_VEL
LIN {X 0,Y 242.266,Z 290.706,A -85,B 0,C 180,E1 -19698.285,E2 -19698.285} C_VEL
LIN {X 0,Y 239.439,Z 278.075,A -85,B 0,C 180,E1 -19699.858,E2 -19699.858} C_VEL
LIN {X 0,Y 235.829,Z 265.351,A -85,B 0,C 180,E1 -19701.179,E2 -19701.179} C_VEL
LIN {X 0,Y 234.344,Z 260.047,A -85,B 0,C 180,E1 -19701.663,E2 -19701.663} C_VEL
LIN {X 0,Y 234.488,Z 259.277,A -85,B 0,C 180,E1 -19703.116,E2 -19703.116} C_VEL
LIN {X 0,Y 234.869,Z 259.228,A -85,B 0,C 180,E1 -19706.571,E2 -19706.571} C_VEL
LIN {X 0,Y 235.593,Z 259.137,A -85,B 0,C 180,E1 -19710.002,E2 -19710.002} C_VEL
LIN {X 0,Y 235.584,Z 259.14,A -85,B 0,C 180,E1 -19711.711,E2 -19711.711} C_VEL
LIN {X 0,Y 235.392,Z 259.164,A -85,B 0,C 180,E1 -19716.861,E2 -19716.861} C_VEL
LIN {X 0,Y 235.227,Z 259.182,A -85,B 0,C 180,E1 -19720.329,E2 -19720.329} C_VEL
LIN {X 0,Y 235.103,Z 259.199,A -85,B 0,C 180,E1 -19725.609,E2 -19725.609} C_VEL
LIN {X 0,Y 235.02,Z 259.212,A -85,B 0,C 180,E1 -19729.206,E2 -19729.206} C_VEL
LIN {X 0,Y 234.98,Z 259.212,A -85,B 0,C 180,E1 -19732.883,E2 -19732.883} C_VEL
LIN {X 0,Y 234.961,Z 259.221,A -85,B 0,C 180,E1 -19736.66,E2 -19736.66} C_VEL
LIN {X 0,Y 234.925,Z 259.224,A -85,B 0,C 180,E1 -19740.571,E2 -19740.571} C_VEL
LIN {X 0,Y 234.954,Z 259.219,A -85,B 0,C 180,E1 -19744.636,E2 -19744.636} C_VEL
LIN {X 0,Y 234.961,Z 259.216,A -85,B 0,C 180,E1 -19748.955,E2 -19748.955} C_VEL
LIN {X 0,Y 234.961,Z 259.215,A -85,B 0,C 180,E1 -19753.471,E2 -19753.471} C_VEL
LIN {X 0,Y 234.956,Z 259.217,A -85,B 0,C 180,E1 -19756.534,E2 -19756.534} C_VEL
LIN {X 0,Y 234.953,Z 259.214,A -85,B 0,C 180,E1 -19761.09,E2 -19761.09} C_VEL
LIN {X 0,Y 234.959,Z 259.201,A -85,B 0,C 180,E1 -19765.371,E2 -19765.371} C_VEL
LIN {X 0,Y 234.969,Z 259.214,A -85,B 0,C 180,E1 -19770.161,E2 -19770.161} C_VEL
LIN {X 0,Y 234.995,Z 259.212,A -85,B 0,C 180,E1 -19773.797,E2 -19773.797} C_VEL
LIN {X 0,Y 235.014,Z 259.195,A -85,B 0,C 180,E1 -19778.973,E2 -19778.973} C_VEL
LIN {X 0,Y 235.1,Z 259.193,A -85,B 0,C 180,E1 -19783.063,E2 -19783.063} C_VEL
LIN {X 0,Y 235.148,Z 259.195,A -85,B 0,C 180,E1 -19787.927,E2 -19787.927} C_VEL
LIN {X 0,Y 235.331,Z 259.166,A -85,B 0,C 180,E1 -19791.415,E2 -19791.415} C_VEL
LIN {X 0,Y 235.373,Z 259.154,A -85,B 0,C 180,E1 -19793.143,E2 -19793.143} C_VEL
LIN {X 0,Y 235.602,Z 259.135,A -85,B 0,C 180,E1 -19798.293,E2 -19798.293} C_VEL
LIN {X 0,Y 235.601,Z 259.139,A -85,B 0,C 180,E1 -19801.712,E2 -19801.712} C_VEL
LIN {X 0,Y 235.37,Z 259.155,A -85,B 0,C 180,E1 -19806.862,E2 -19806.862} C_VEL
LIN {X 0,Y 235.222,Z 259.18,A -85,B 0,C 180,E1 -19810.33,E2 -19810.33} C_VEL
LIN {X 0,Y 235.124,Z 259.196,A -85,B 0,C 180,E1 -19815.608,E2 -19815.608} C_VEL
LIN {X 0,Y 235.019,Z 259.202,A -85,B 0,C 180,E1 -19819.207,E2 -19819.207} C_VEL
LIN {X 0,Y 234.972,Z 259.215,A -85,B 0,C 180,E1 -19822.884,E2 -19822.884} C_VEL
LIN {X 0,Y 234.979,Z 259.211,A -85,B 0,C 180,E1 -19826.659,E2 -19826.659} C_VEL
LIN {X 0,Y 234.933,Z 259.219,A -85,B 0,C 180,E1 -19830.57,E2 -19830.57} C_VEL
LIN {X 0,Y 234.938,Z 259.219,A -85,B 0,C 180,E1 -19834.639,E2 -19834.639} C_VEL
LIN {X 0,Y 235.003,Z 259.378,A -85,B 0,C 180,E1 -19839.155,E2 -19839.155} C_VEL
LIN {X 0,Y 235.685,Z 263.348,A -85,B 0,C 180,E1 -19843.305,E2 -19843.305} C_VEL
